// ---- DUTs/IO/Boxes/EP2008_E2806B95.TcDUT
{attribute 'GeneratedUsingTerminal: EP2008-0001-0016'}
{attribute addProperty BoxType "EP2008-0001-0016"}
{attribute addProperty Description "EP2008-0001 8 Ch. Dig. Output 24V, 0,5A, M8"}
{attribute addProperty Physics "YY"}
{attribute addProperty Id "Channel_1AT %Q*Channel_42CA91F71Channel_2AT %Q*Channel_42CA91F71Channel_3AT %Q*Channel_42CA91F71Channel_4AT %Q*Channel_42CA91F71Channel_5AT %Q*Channel_42CA91F71Channel_6AT %Q*Channel_42CA91F71Channel_7AT %Q*Channel_42CA91F71Channel_8AT %Q*Channel_42CA91F71WcStateAT %I*WcState_0B2B16F91InfoDataAT %I*InfoData_6F19DB2B2"}
{attribute addProperty CRC "3800066965"}
{attribute addProperty Size "11"}
TYPE EP2008_E2806B95 EXTENDS EtcSlaveBoxBase_77A0E4A7 :
STRUCT
	{attribute addProperty Name "Channel_1"}
	Channel_1 : Channel_42CA91F7;
	{attribute addProperty Name "Channel_2"}
	Channel_2 : Channel_42CA91F7;
	{attribute addProperty Name "Channel_3"}
	Channel_3 : Channel_42CA91F7;
	{attribute addProperty Name "Channel_4"}
	Channel_4 : Channel_42CA91F7;
	{attribute addProperty Name "Channel_5"}
	Channel_5 : Channel_42CA91F7;
	{attribute addProperty Name "Channel_6"}
	Channel_6 : Channel_42CA91F7;
	{attribute addProperty Name "Channel_7"}
	Channel_7 : Channel_42CA91F7;
	{attribute addProperty Name "Channel_8"}
	Channel_8 : Channel_42CA91F7;
	{attribute addProperty Name "WcState"}
	WcState : WcState_0B2B16F9;
	{attribute addProperty Name "InfoData"}
	InfoData : InfoData_6F19DB2B;
END_STRUCT
END_TYPE

// ---- DUTs/IO/Boxes/EP2028_E2806B95.TcDUT
{attribute 'GeneratedUsingTerminal: EP2028-0001-0016'}
{attribute addProperty BoxType "EP2028-0001-0016"}
{attribute addProperty Description "EP2028-0001 8 Ch. Dig. Output 24V, 2A, M8"}
{attribute addProperty Physics "YY"}
{attribute addProperty Id "Channel_1AT %Q*Channel_42CA91F71Channel_2AT %Q*Channel_42CA91F71Channel_3AT %Q*Channel_42CA91F71Channel_4AT %Q*Channel_42CA91F71Channel_5AT %Q*Channel_42CA91F71Channel_6AT %Q*Channel_42CA91F71Channel_7AT %Q*Channel_42CA91F71Channel_8AT %Q*Channel_42CA91F71WcStateAT %I*WcState_0B2B16F91InfoDataAT %I*InfoData_6F19DB2B2"}
{attribute addProperty CRC "3800066965"}
{attribute addProperty Size "11"}
TYPE EP2028_E2806B95 EXTENDS EtcSlaveBoxBase_77A0E4A7 :
STRUCT
	{attribute addProperty Name "Channel_1"}
	Channel_1 : Channel_42CA91F7;
	{attribute addProperty Name "Channel_2"}
	Channel_2 : Channel_42CA91F7;
	{attribute addProperty Name "Channel_3"}
	Channel_3 : Channel_42CA91F7;
	{attribute addProperty Name "Channel_4"}
	Channel_4 : Channel_42CA91F7;
	{attribute addProperty Name "Channel_5"}
	Channel_5 : Channel_42CA91F7;
	{attribute addProperty Name "Channel_6"}
	Channel_6 : Channel_42CA91F7;
	{attribute addProperty Name "Channel_7"}
	Channel_7 : Channel_42CA91F7;
	{attribute addProperty Name "Channel_8"}
	Channel_8 : Channel_42CA91F7;
	{attribute addProperty Name "WcState"}
	WcState : WcState_0B2B16F9;
	{attribute addProperty Name "InfoData"}
	InfoData : InfoData_6F19DB2B;
END_STRUCT
END_TYPE

// ---- DUTs/IO/Boxes/EP2038_3AE10DD7.TcDUT
{attribute 'GeneratedUsingTerminal: EP2038-0001-0016'}
{attribute addProperty BoxType "EP2038-0001-0016"}
{attribute addProperty Description "EP2038-0001 8 Ch. Dig. Output 24V, 2A, M8, Diagnostic"}
{attribute addProperty Physics "YY"}
{attribute addProperty Id "Diag_Channel_1AT %I*Diag_Channel_830843C11Diag_Channel_2AT %I*Diag_Channel_830843C11Diag_Channel_3AT %I*Diag_Channel_830843C11Diag_Channel_4AT %I*Diag_Channel_830843C11Diag_Channel_5AT %I*Diag_Channel_830843C11Diag_Channel_6AT %I*Diag_Channel_830843C11Diag_Channel_7AT %I*Diag_Channel_830843C11Diag_Channel_8AT %I*Diag_Channel_830843C11Channel_1AT %Q*Channel_42CA91F71Channel_2AT %Q*Channel_42CA91F71Channel_3AT %Q*Channel_42CA91F71Channel_4AT %Q*Channel_42CA91F71Channel_5AT %Q*Channel_42CA91F71Channel_6AT %Q*Channel_42CA91F71Channel_7AT %Q*Channel_42CA91F71Channel_8AT %Q*Channel_42CA91F71WcStateAT %I*WcState_9091E0EB2InfoDataAT %I*InfoData_6F19DB2B2"}
{attribute addProperty CRC "987827671"}
{attribute addProperty Size "20"}
TYPE EP2038_3AE10DD7 EXTENDS EtcSlaveBoxBase_77A0E4A7 :
STRUCT
	{attribute addProperty Name "Diag_Channel_1"}
	Diag_Channel_1 : Diag_Channel_830843C1;
	{attribute addProperty Name "Diag_Channel_2"}
	Diag_Channel_2 : Diag_Channel_830843C1;
	{attribute addProperty Name "Diag_Channel_3"}
	Diag_Channel_3 : Diag_Channel_830843C1;
	{attribute addProperty Name "Diag_Channel_4"}
	Diag_Channel_4 : Diag_Channel_830843C1;
	{attribute addProperty Name "Diag_Channel_5"}
	Diag_Channel_5 : Diag_Channel_830843C1;
	{attribute addProperty Name "Diag_Channel_6"}
	Diag_Channel_6 : Diag_Channel_830843C1;
	{attribute addProperty Name "Diag_Channel_7"}
	Diag_Channel_7 : Diag_Channel_830843C1;
	{attribute addProperty Name "Diag_Channel_8"}
	Diag_Channel_8 : Diag_Channel_830843C1;
	{attribute addProperty Name "Channel_1"}
	Channel_1 : Channel_42CA91F7;
	{attribute addProperty Name "Channel_2"}
	Channel_2 : Channel_42CA91F7;
	{attribute addProperty Name "Channel_3"}
	Channel_3 : Channel_42CA91F7;
	{attribute addProperty Name "Channel_4"}
	Channel_4 : Channel_42CA91F7;
	{attribute addProperty Name "Channel_5"}
	Channel_5 : Channel_42CA91F7;
	{attribute addProperty Name "Channel_6"}
	Channel_6 : Channel_42CA91F7;
	{attribute addProperty Name "Channel_7"}
	Channel_7 : Channel_42CA91F7;
	{attribute addProperty Name "Channel_8"}
	Channel_8 : Channel_42CA91F7;
	{attribute addProperty Name "WcState"}
	WcState : WcState_9091E0EB;
	{attribute addProperty Name "InfoData"}
	InfoData : InfoData_6F19DB2B;
END_STRUCT
END_TYPE

// ---- DUTs/IO/Boxes/EP2308_F6D9A8D1.TcDUT
{attribute 'GeneratedUsingTerminal: EP2308-0000-0016'}
{attribute addProperty BoxType "EP2308-0000-0016"}
{attribute addProperty Description "EP2308-0000 4 Ch. Dig. In, 3ms, 4 Ch. Dig. Out 24V, 0,5A, S8"}
{attribute addProperty Physics "YY"}
{attribute addProperty Id "Channel_1AT %I*Channel_830843C11Channel_2AT %I*Channel_830843C11Channel_3AT %I*Channel_830843C11Channel_4AT %I*Channel_830843C11Channel_5AT %Q*Channel_42CA91F71Channel_6AT %Q*Channel_42CA91F71Channel_7AT %Q*Channel_42CA91F71Channel_8AT %Q*Channel_42CA91F71WcStateAT %I*WcState_9091E0EB2InfoDataAT %I*InfoData_6F19DB2B2"}
{attribute addProperty CRC "4141459665"}
{attribute addProperty Size "12"}
TYPE EP2308_F6D9A8D1 EXTENDS EtcSlaveBoxBase_77A0E4A7 :
STRUCT
	{attribute addProperty Name "Channel_1"}
	Channel_1 : Channel_830843C1;
	{attribute addProperty Name "Channel_2"}
	Channel_2 : Channel_830843C1;
	{attribute addProperty Name "Channel_3"}
	Channel_3 : Channel_830843C1;
	{attribute addProperty Name "Channel_4"}
	Channel_4 : Channel_830843C1;
	{attribute addProperty Name "Channel_5"}
	Channel_5 : Channel_42CA91F7;
	{attribute addProperty Name "Channel_6"}
	Channel_6 : Channel_42CA91F7;
	{attribute addProperty Name "Channel_7"}
	Channel_7 : Channel_42CA91F7;
	{attribute addProperty Name "Channel_8"}
	Channel_8 : Channel_42CA91F7;
	{attribute addProperty Name "WcState"}
	WcState : WcState_9091E0EB;
	{attribute addProperty Name "InfoData"}
	InfoData : InfoData_6F19DB2B;
END_STRUCT
END_TYPE

// ---- DUTs/IO/Boxes/EP2316_CAC4656D.TcDUT
{attribute 'GeneratedUsingTerminal: EP2316-0003-0016'}
{attribute addProperty BoxType "EP2316-0003-0016"}
{attribute addProperty Description "EP2316-0003 8 Ch. Dig. In, 10µs, 8Ch. Dig. Out 24V, 0,5A, Diagnostic, 10-Pole Plug Connector"}
{attribute addProperty Physics "YY"}
{attribute addProperty Id "DIG_InputsAT %I*DIG_Inputs_CC4551489DIG_Diag_InputsAT %I*DIG_Diag_Inputs_584303BF8DIG_Inputs_DeviceAT %I*DIG_Inputs_Device_E94E5BF95DIG_OutputsAT %Q*DIG_Outputs_28AC1A9E8DIG_Outputs_DeviceAT %Q*DIG_Outputs_Device_36A5EF172WcStateAT %I*WcState_9091E0EB2InfoDataAT %I*InfoData_32EB74EA10"}
{attribute addProperty CRC "3401868653"}
{attribute addProperty Size "44"}
TYPE EP2316_CAC4656D EXTENDS EtcSlaveBoxBase_77A0E4A7 :
STRUCT
	{attribute addProperty Name "DIG_Inputs"}
	DIG_Inputs : DIG_Inputs_CC455148;
	{attribute addProperty Name "DIG_Diag_Inputs"}
	DIG_Diag_Inputs : DIG_Diag_Inputs_584303BF;
	{attribute addProperty Name "DIG_Inputs_Device"}
	DIG_Inputs_Device : DIG_Inputs_Device_E94E5BF9;
	{attribute addProperty Name "DIG_Outputs"}
	DIG_Outputs : DIG_Outputs_28AC1A9E;
	{attribute addProperty Name "DIG_Outputs_Device"}
	DIG_Outputs_Device : DIG_Outputs_Device_36A5EF17;
	{attribute addProperty Name "WcState"}
	WcState : WcState_9091E0EB;
	{attribute addProperty Name "InfoData"}
	InfoData : InfoData_32EB74EA;
END_STRUCT
END_TYPE

// ---- DUTs/IO/Boxes/EP2316_528F6B1F.TcDUT
{attribute 'GeneratedUsingTerminal: EP2316-0008-0016'}
{attribute addProperty BoxType "EP2316-0008-0016"}
{attribute addProperty Description "EP2316-0008 8 Ch. Dig. In, 10µs, 8Ch. Dig. Out 24V, 0,5A, Diagnostic, D-SUB25"}
{attribute addProperty Physics "YY"}
{attribute addProperty Id "DO_InputsAT %I*DO_Inputs_CC4551489DO_Diag_InputsAT %I*DO_Diag_Inputs_584303BF8DO_Inputs_DeviceAT %I*DO_Inputs_Device_AF161A9E4DO_OutputsAT %Q*DO_Outputs_28AC1A9E8DO_Outputs_DeviceAT %Q*DO_Outputs_Device_36A5EF172WcStateAT %I*WcState_9091E0EB2InfoDataAT %I*InfoData_32EB74EA10"}
{attribute addProperty CRC "1385130783"}
{attribute addProperty Size "43"}
TYPE EP2316_528F6B1F EXTENDS EtcSlaveBoxBase_77A0E4A7 :
STRUCT
	{attribute addProperty Name "DO_Inputs"}
	DO_Inputs : DO_Inputs_CC455148;
	{attribute addProperty Name "DO_Diag_Inputs"}
	DO_Diag_Inputs : DO_Diag_Inputs_584303BF;
	{attribute addProperty Name "DO_Inputs_Device"}
	DO_Inputs_Device : DO_Inputs_Device_AF161A9E;
	{attribute addProperty Name "DO_Outputs"}
	DO_Outputs : DO_Outputs_28AC1A9E;
	{attribute addProperty Name "DO_Outputs_Device"}
	DO_Outputs_Device : DO_Outputs_Device_36A5EF17;
	{attribute addProperty Name "WcState"}
	WcState : WcState_9091E0EB;
	{attribute addProperty Name "InfoData"}
	InfoData : InfoData_32EB74EA;
END_STRUCT
END_TYPE

// ---- DUTs/IO/Boxes/EP2316_3C060514.TcDUT
{attribute 'GeneratedUsingTerminal: EP2316-0008-0017'}
{attribute addProperty BoxType "EP2316-0008-0017"}
{attribute addProperty Description "EP2316-0008 8 Ch. Dig. In, 10µs, 8Ch. Dig. Out 24V, 0,5A, Diagnostic, D-SUB25"}
{attribute addProperty Physics "YY"}
{attribute addProperty Id "DO_Diag_InputsAT %I*DO_Diag_Inputs_CC4551489DO_Diag_Inputs_1AT %I*DO_Diag_Inputs_212B82C19DO_Inputs_DeviceAT %I*DO_Inputs_Device_AF161A9E4DO_OutputsAT %Q*DO_Outputs_28AC1A9E8DO_Outputs_DeviceAT %Q*DO_Outputs_Device_36A5EF172WcStateAT %I*WcState_9091E0EB2InfoDataAT %I*InfoData_32EB74EA10"}
{attribute addProperty CRC "1007027476"}
{attribute addProperty Size "44"}
TYPE EP2316_3C060514 EXTENDS EtcSlaveBoxBase_77A0E4A7 :
STRUCT
	{attribute addProperty Name "DO_Diag_Inputs"}
	DO_Diag_Inputs : DO_Diag_Inputs_CC455148;
	{attribute addProperty Name "DO_Diag_Inputs_1"}
	DO_Diag_Inputs_1 : DO_Diag_Inputs_212B82C1;
	{attribute addProperty Name "DO_Inputs_Device"}
	DO_Inputs_Device : DO_Inputs_Device_AF161A9E;
	{attribute addProperty Name "DO_Outputs"}
	DO_Outputs : DO_Outputs_28AC1A9E;
	{attribute addProperty Name "DO_Outputs_Device"}
	DO_Outputs_Device : DO_Outputs_Device_36A5EF17;
	{attribute addProperty Name "WcState"}
	WcState : WcState_9091E0EB;
	{attribute addProperty Name "InfoData"}
	InfoData : InfoData_32EB74EA;
END_STRUCT
END_TYPE

// ---- DUTs/IO/Boxes/EP2316_DCD24F8F.TcDUT
{attribute 'GeneratedUsingTerminal: EP2316-0008-0018'}
{attribute addProperty BoxType "EP2316-0008-0018"}
{attribute addProperty Description "EP2316-0008 8 Ch. Dig. In, 10µs, 8Ch. Dig. Out 24V, 0,5A, Diagnostic, D-SUB25"}
{attribute addProperty Physics "YY"}
{attribute addProperty Id "DIG_InputsAT %I*DIG_Inputs_CC4551489DIG_Diag_InputsAT %I*DIG_Diag_Inputs_584303BF8DIG_Inputs_DeviceAT %I*DIG_Inputs_Device_4E5AF17E5DIG_OutputsAT %Q*DIG_Outputs_28AC1A9E8DIG_Outputs_DeviceAT %Q*DIG_Outputs_Device_36A5EF172WcStateAT %I*WcState_9091E0EB2InfoDataAT %I*InfoData_32EB74EA10"}
{attribute addProperty CRC "3704770447"}
{attribute addProperty Size "44"}
TYPE EP2316_DCD24F8F EXTENDS EtcSlaveBoxBase_77A0E4A7 :
STRUCT
	{attribute addProperty Name "DIG_Inputs"}
	DIG_Inputs : DIG_Inputs_CC455148;
	{attribute addProperty Name "DIG_Diag_Inputs"}
	DIG_Diag_Inputs : DIG_Diag_Inputs_584303BF;
	{attribute addProperty Name "DIG_Inputs_Device"}
	DIG_Inputs_Device : DIG_Inputs_Device_4E5AF17E;
	{attribute addProperty Name "DIG_Outputs"}
	DIG_Outputs : DIG_Outputs_28AC1A9E;
	{attribute addProperty Name "DIG_Outputs_Device"}
	DIG_Outputs_Device : DIG_Outputs_Device_36A5EF17;
	{attribute addProperty Name "WcState"}
	WcState : WcState_9091E0EB;
	{attribute addProperty Name "InfoData"}
	InfoData : InfoData_32EB74EA;
END_STRUCT
END_TYPE

// ---- DUTs/IO/Boxes/EP2318_F6D9A8D1.TcDUT
{attribute 'GeneratedUsingTerminal: EP2318-0001-0016'}
{attribute addProperty BoxType "EP2318-0001-0016"}
{attribute addProperty Description "EP2318-0001 4 Ch. Dig. In, 10µs, 4 Ch. Dig. Out 24V, 0,5A, M8"}
{attribute addProperty Physics "YY"}
{attribute addProperty Id "Channel_1AT %I*Channel_830843C11Channel_2AT %I*Channel_830843C11Channel_3AT %I*Channel_830843C11Channel_4AT %I*Channel_830843C11Channel_5AT %Q*Channel_42CA91F71Channel_6AT %Q*Channel_42CA91F71Channel_7AT %Q*Channel_42CA91F71Channel_8AT %Q*Channel_42CA91F71WcStateAT %I*WcState_9091E0EB2InfoDataAT %I*InfoData_6F19DB2B2"}
{attribute addProperty CRC "4141459665"}
{attribute addProperty Size "12"}
TYPE EP2318_F6D9A8D1 EXTENDS EtcSlaveBoxBase_77A0E4A7 :
STRUCT
	{attribute addProperty Name "Channel_1"}
	Channel_1 : Channel_830843C1;
	{attribute addProperty Name "Channel_2"}
	Channel_2 : Channel_830843C1;
	{attribute addProperty Name "Channel_3"}
	Channel_3 : Channel_830843C1;
	{attribute addProperty Name "Channel_4"}
	Channel_4 : Channel_830843C1;
	{attribute addProperty Name "Channel_5"}
	Channel_5 : Channel_42CA91F7;
	{attribute addProperty Name "Channel_6"}
	Channel_6 : Channel_42CA91F7;
	{attribute addProperty Name "Channel_7"}
	Channel_7 : Channel_42CA91F7;
	{attribute addProperty Name "Channel_8"}
	Channel_8 : Channel_42CA91F7;
	{attribute addProperty Name "WcState"}
	WcState : WcState_9091E0EB;
	{attribute addProperty Name "InfoData"}
	InfoData : InfoData_6F19DB2B;
END_STRUCT
END_TYPE

// ---- DUTs/IO/Boxes/EP2328_F6D9A8D1.TcDUT
{attribute 'GeneratedUsingTerminal: EP2328-0001-0016'}
{attribute addProperty BoxType "EP2328-0001-0016"}
{attribute addProperty Description "EP2328-0001 4 CH. Dig. In, 3ms, 4 Ch. Dig. Out 24V, 2A, M8"}
{attribute addProperty Physics "YY"}
{attribute addProperty Id "Channel_1AT %I*Channel_830843C11Channel_2AT %I*Channel_830843C11Channel_3AT %I*Channel_830843C11Channel_4AT %I*Channel_830843C11Channel_5AT %Q*Channel_42CA91F71Channel_6AT %Q*Channel_42CA91F71Channel_7AT %Q*Channel_42CA91F71Channel_8AT %Q*Channel_42CA91F71WcStateAT %I*WcState_9091E0EB2InfoDataAT %I*InfoData_6F19DB2B2"}
{attribute addProperty CRC "4141459665"}
{attribute addProperty Size "12"}
TYPE EP2328_F6D9A8D1 EXTENDS EtcSlaveBoxBase_77A0E4A7 :
STRUCT
	{attribute addProperty Name "Channel_1"}
	Channel_1 : Channel_830843C1;
	{attribute addProperty Name "Channel_2"}
	Channel_2 : Channel_830843C1;
	{attribute addProperty Name "Channel_3"}
	Channel_3 : Channel_830843C1;
	{attribute addProperty Name "Channel_4"}
	Channel_4 : Channel_830843C1;
	{attribute addProperty Name "Channel_5"}
	Channel_5 : Channel_42CA91F7;
	{attribute addProperty Name "Channel_6"}
	Channel_6 : Channel_42CA91F7;
	{attribute addProperty Name "Channel_7"}
	Channel_7 : Channel_42CA91F7;
	{attribute addProperty Name "Channel_8"}
	Channel_8 : Channel_42CA91F7;
	{attribute addProperty Name "WcState"}
	WcState : WcState_9091E0EB;
	{attribute addProperty Name "InfoData"}
	InfoData : InfoData_6F19DB2B;
END_STRUCT
END_TYPE

// ---- DUTs/IO/Boxes/EP2328_F66CDDB7.TcDUT
{attribute 'GeneratedUsingTerminal: EP2328-1061-0016'}
{attribute addProperty BoxType "EP2328-1061-0016"}
{attribute addProperty Description "EP2328-1061 4 Ch. Dig. In, 10µs, 4 Ch. Dig. Out 24V, 2A, M8 cable"}
{attribute addProperty Physics "YY"}
{attribute addProperty Id "DI_X01_Pin4_InputAT %I*DI_X01_Pin4_Input_830843C11DI_X01_Pin2_InputAT %I*DI_X01_Pin2_Input_830843C11DI_X02_Pin4_InputAT %I*DI_X02_Pin4_Input_830843C11DI_X02_Pin2_InputAT %I*DI_X02_Pin2_Input_830843C11DO_X03_Pin4_OutputAT %Q*DO_X03_Pin4_Output_42CA91F71DO_X03_Pin2_OutputAT %Q*DO_X03_Pin2_Output_42CA91F71DO_X04_Pin4_OutputAT %Q*DO_X04_Pin4_Output_42CA91F71DO_X04_Pin2_OutputAT %Q*DO_X04_Pin2_Output_42CA91F71WcStateAT %I*WcState_9091E0EB2InfoDataAT %I*InfoData_6F19DB2B2"}
{attribute addProperty CRC "4134329783"}
{attribute addProperty Size "12"}
TYPE EP2328_F66CDDB7 EXTENDS EtcSlaveBoxBase_77A0E4A7 :
STRUCT
	{attribute addProperty Name "DI_X01_Pin4_Input"}
	DI_X01_Pin4_Input : DI_X01_Pin4_Input_830843C1;
	{attribute addProperty Name "DI_X01_Pin2_Input"}
	DI_X01_Pin2_Input : DI_X01_Pin2_Input_830843C1;
	{attribute addProperty Name "DI_X02_Pin4_Input"}
	DI_X02_Pin4_Input : DI_X02_Pin4_Input_830843C1;
	{attribute addProperty Name "DI_X02_Pin2_Input"}
	DI_X02_Pin2_Input : DI_X02_Pin2_Input_830843C1;
	{attribute addProperty Name "DO_X03_Pin4_Output"}
	DO_X03_Pin4_Output : DO_X03_Pin4_Output_42CA91F7;
	{attribute addProperty Name "DO_X03_Pin2_Output"}
	DO_X03_Pin2_Output : DO_X03_Pin2_Output_42CA91F7;
	{attribute addProperty Name "DO_X04_Pin4_Output"}
	DO_X04_Pin4_Output : DO_X04_Pin4_Output_42CA91F7;
	{attribute addProperty Name "DO_X04_Pin2_Output"}
	DO_X04_Pin2_Output : DO_X04_Pin2_Output_42CA91F7;
	{attribute addProperty Name "WcState"}
	WcState : WcState_9091E0EB;
	{attribute addProperty Name "InfoData"}
	InfoData : InfoData_6F19DB2B;
END_STRUCT
END_TYPE

// ---- DUTs/IO/Boxes/EP2338_39FFBC52.TcDUT
{attribute 'GeneratedUsingTerminal: EP2338-0001-0016'}
{attribute addProperty BoxType "EP2338-0001-0016"}
{attribute addProperty Description "EP2338-0001 8 Ch. Dig. Input/Output 24V, 0,5A, M8"}
{attribute addProperty Physics "YY"}
{attribute addProperty Id "Channel_1AT %I*Channel_830843C11Channel_2AT %I*Channel_830843C11Channel_3AT %I*Channel_830843C11Channel_4AT %I*Channel_830843C11Channel_5AT %I*Channel_830843C11Channel_6AT %I*Channel_830843C11Channel_7AT %I*Channel_830843C11Channel_8AT %I*Channel_830843C11Channel_1_1AT %Q*Channel_42CA91F71Channel_2_1AT %Q*Channel_42CA91F71Channel_3_1AT %Q*Channel_42CA91F71Channel_4_1AT %Q*Channel_42CA91F71Channel_5_1AT %Q*Channel_42CA91F71Channel_6_1AT %Q*Channel_42CA91F71Channel_7_1AT %Q*Channel_42CA91F71Channel_8_1AT %Q*Channel_42CA91F71WcStateAT %I*WcState_9091E0EB2InfoDataAT %I*InfoData_6F19DB2B2"}
{attribute addProperty CRC "973061202"}
{attribute addProperty Size "20"}
TYPE EP2338_39FFBC52 EXTENDS EtcSlaveBoxBase_77A0E4A7 :
STRUCT
	{attribute addProperty Name "Channel_1"}
	Channel_1 : Channel_830843C1;
	{attribute addProperty Name "Channel_2"}
	Channel_2 : Channel_830843C1;
	{attribute addProperty Name "Channel_3"}
	Channel_3 : Channel_830843C1;
	{attribute addProperty Name "Channel_4"}
	Channel_4 : Channel_830843C1;
	{attribute addProperty Name "Channel_5"}
	Channel_5 : Channel_830843C1;
	{attribute addProperty Name "Channel_6"}
	Channel_6 : Channel_830843C1;
	{attribute addProperty Name "Channel_7"}
	Channel_7 : Channel_830843C1;
	{attribute addProperty Name "Channel_8"}
	Channel_8 : Channel_830843C1;
	{attribute addProperty Name "Channel_1_1"}
	Channel_1_1 : Channel_42CA91F7;
	{attribute addProperty Name "Channel_2_1"}
	Channel_2_1 : Channel_42CA91F7;
	{attribute addProperty Name "Channel_3_1"}
	Channel_3_1 : Channel_42CA91F7;
	{attribute addProperty Name "Channel_4_1"}
	Channel_4_1 : Channel_42CA91F7;
	{attribute addProperty Name "Channel_5_1"}
	Channel_5_1 : Channel_42CA91F7;
	{attribute addProperty Name "Channel_6_1"}
	Channel_6_1 : Channel_42CA91F7;
	{attribute addProperty Name "Channel_7_1"}
	Channel_7_1 : Channel_42CA91F7;
	{attribute addProperty Name "Channel_8_1"}
	Channel_8_1 : Channel_42CA91F7;
	{attribute addProperty Name "WcState"}
	WcState : WcState_9091E0EB;
	{attribute addProperty Name "InfoData"}
	InfoData : InfoData_6F19DB2B;
END_STRUCT
END_TYPE

// ---- DUTs/IO/Boxes/EP2338_7699BCF6.TcDUT
{attribute 'GeneratedUsingTerminal: EP2338-0001-0018'}
{attribute addProperty BoxType "EP2338-0001-0018"}
{attribute addProperty Description "EP2338-0001 8 Ch. Dig. Input/Output 24V, 0,5A, M8"}
{attribute addProperty Physics "YY"}
{attribute addProperty Id "Channel_1AT %I*Channel_830843C11Channel_2AT %I*Channel_830843C11Channel_3AT %I*Channel_830843C11Channel_4AT %I*Channel_830843C11Channel_5AT %I*Channel_830843C11Channel_6AT %I*Channel_830843C11Channel_7AT %I*Channel_830843C11Channel_8AT %I*Channel_830843C11Channel_9AT %Q*Channel_42CA91F71Channel_10AT %Q*Channel_42CA91F71Channel_11AT %Q*Channel_42CA91F71Channel_12AT %Q*Channel_42CA91F71Channel_13AT %Q*Channel_42CA91F71Channel_14AT %Q*Channel_42CA91F71Channel_15AT %Q*Channel_42CA91F71Channel_16AT %Q*Channel_42CA91F71WcStateAT %I*WcState_9091E0EB2InfoDataAT %I*InfoData_6F19DB2B2"}
{attribute addProperty CRC "1989786870"}
{attribute addProperty Size "20"}
TYPE EP2338_7699BCF6 EXTENDS EtcSlaveBoxBase_77A0E4A7 :
STRUCT
	{attribute addProperty Name "Channel_1"}
	Channel_1 : Channel_830843C1;
	{attribute addProperty Name "Channel_2"}
	Channel_2 : Channel_830843C1;
	{attribute addProperty Name "Channel_3"}
	Channel_3 : Channel_830843C1;
	{attribute addProperty Name "Channel_4"}
	Channel_4 : Channel_830843C1;
	{attribute addProperty Name "Channel_5"}
	Channel_5 : Channel_830843C1;
	{attribute addProperty Name "Channel_6"}
	Channel_6 : Channel_830843C1;
	{attribute addProperty Name "Channel_7"}
	Channel_7 : Channel_830843C1;
	{attribute addProperty Name "Channel_8"}
	Channel_8 : Channel_830843C1;
	{attribute addProperty Name "Channel_9"}
	Channel_9 : Channel_42CA91F7;
	{attribute addProperty Name "Channel_10"}
	Channel_10 : Channel_42CA91F7;
	{attribute addProperty Name "Channel_11"}
	Channel_11 : Channel_42CA91F7;
	{attribute addProperty Name "Channel_12"}
	Channel_12 : Channel_42CA91F7;
	{attribute addProperty Name "Channel_13"}
	Channel_13 : Channel_42CA91F7;
	{attribute addProperty Name "Channel_14"}
	Channel_14 : Channel_42CA91F7;
	{attribute addProperty Name "Channel_15"}
	Channel_15 : Channel_42CA91F7;
	{attribute addProperty Name "Channel_16"}
	Channel_16 : Channel_42CA91F7;
	{attribute addProperty Name "WcState"}
	WcState : WcState_9091E0EB;
	{attribute addProperty Name "InfoData"}
	InfoData : InfoData_6F19DB2B;
END_STRUCT
END_TYPE

// ---- DUTs/IO/Boxes/EP2339_B2B612E8.TcDUT
{attribute 'GeneratedUsingTerminal: EP2339-0003-0016'}
{attribute addProperty BoxType "EP2339-0003-0016"}
{attribute addProperty Description "EP2339-0003 16 Ch. Dig. Input/Output 24V, 0,5A, 10-Pole Plug Connector"}
{attribute addProperty Physics "YY"}
{attribute addProperty Id "DI_Inputs_Channel_1AT %I*DI_Inputs_Channel_91AC31B711DI_Inputs_Channel_2AT %I*DI_Inputs_Channel_91AC31B711DO_Outputs_Channel_1AT %Q*DO_Outputs_Channel_28AC1A9E8DO_Outputs_Channel_2AT %Q*DO_Outputs_Channel_28AC1A9E8WcStateAT %I*WcState_9091E0EB2InfoDataAT %I*InfoData_32EB74EA10"}
{attribute addProperty CRC "2998276840"}
{attribute addProperty Size "50"}
TYPE EP2339_B2B612E8 EXTENDS EtcSlaveBoxBase_77A0E4A7 :
STRUCT
	{attribute addProperty Name "DI_Inputs_Channel_1"}
	DI_Inputs_Channel_1 : DI_Inputs_Channel_91AC31B7;
	{attribute addProperty Name "DI_Inputs_Channel_2"}
	DI_Inputs_Channel_2 : DI_Inputs_Channel_91AC31B7;
	{attribute addProperty Name "DO_Outputs_Channel_1"}
	DO_Outputs_Channel_1 : DO_Outputs_Channel_28AC1A9E;
	{attribute addProperty Name "DO_Outputs_Channel_2"}
	DO_Outputs_Channel_2 : DO_Outputs_Channel_28AC1A9E;
	{attribute addProperty Name "WcState"}
	WcState : WcState_9091E0EB;
	{attribute addProperty Name "InfoData"}
	InfoData : InfoData_32EB74EA;
END_STRUCT
END_TYPE

// ---- DUTs/IO/Boxes/EP2339_C2A6198C.TcDUT
{attribute 'GeneratedUsingTerminal: EP2339-0021-0016'}
{attribute addProperty BoxType "EP2339-0021-0016"}
{attribute addProperty Description "EP2339-0021 16 Ch. Dig. Input/Output 24V, 0,5A, M8"}
{attribute addProperty Physics "YY"}
{attribute addProperty Id "Channel_1AT %I*Channel_830843C11Channel_2AT %I*Channel_830843C11Channel_3AT %I*Channel_830843C11Channel_4AT %I*Channel_830843C11Channel_5AT %I*Channel_830843C11Channel_6AT %I*Channel_830843C11Channel_7AT %I*Channel_830843C11Channel_8AT %I*Channel_830843C11Channel_9AT %I*Channel_830843C11Channel_10AT %I*Channel_830843C11Channel_11AT %I*Channel_830843C11Channel_12AT %I*Channel_830843C11Channel_13AT %I*Channel_830843C11Channel_14AT %I*Channel_830843C11Channel_15AT %I*Channel_830843C11Channel_16AT %I*Channel_830843C11Channel_1_1AT %Q*Channel_42CA91F71Channel_2_1AT %Q*Channel_42CA91F71Channel_3_1AT %Q*Channel_42CA91F71Channel_4_1AT %Q*Channel_42CA91F71Channel_5_1AT %Q*Channel_42CA91F71Channel_6_1AT %Q*Channel_42CA91F71Channel_7_1AT %Q*Channel_42CA91F71Channel_8_1AT %Q*Channel_42CA91F71Channel_9_1AT %Q*Channel_42CA91F71Channel_10_1AT %Q*Channel_42CA91F71Channel_11_1AT %Q*Channel_42CA91F71Channel_12_1AT %Q*Channel_42CA91F71Channel_13_1AT %Q*Channel_42CA91F71Channel_14_1AT %Q*Channel_42CA91F71Channel_15_1AT %Q*Channel_42CA91F71Channel_16_1AT %Q*Channel_42CA91F71WcStateAT %I*WcState_9091E0EB2InfoDataAT %I*InfoData_0A66F0098"}
{attribute addProperty CRC "3265665420"}
{attribute addProperty Size "42"}
TYPE EP2339_C2A6198C EXTENDS EtcSlaveBoxBase_77A0E4A7 :
STRUCT
	{attribute addProperty Name "Channel_1"}
	Channel_1 : Channel_830843C1;
	{attribute addProperty Name "Channel_2"}
	Channel_2 : Channel_830843C1;
	{attribute addProperty Name "Channel_3"}
	Channel_3 : Channel_830843C1;
	{attribute addProperty Name "Channel_4"}
	Channel_4 : Channel_830843C1;
	{attribute addProperty Name "Channel_5"}
	Channel_5 : Channel_830843C1;
	{attribute addProperty Name "Channel_6"}
	Channel_6 : Channel_830843C1;
	{attribute addProperty Name "Channel_7"}
	Channel_7 : Channel_830843C1;
	{attribute addProperty Name "Channel_8"}
	Channel_8 : Channel_830843C1;
	{attribute addProperty Name "Channel_9"}
	Channel_9 : Channel_830843C1;
	{attribute addProperty Name "Channel_10"}
	Channel_10 : Channel_830843C1;
	{attribute addProperty Name "Channel_11"}
	Channel_11 : Channel_830843C1;
	{attribute addProperty Name "Channel_12"}
	Channel_12 : Channel_830843C1;
	{attribute addProperty Name "Channel_13"}
	Channel_13 : Channel_830843C1;
	{attribute addProperty Name "Channel_14"}
	Channel_14 : Channel_830843C1;
	{attribute addProperty Name "Channel_15"}
	Channel_15 : Channel_830843C1;
	{attribute addProperty Name "Channel_16"}
	Channel_16 : Channel_830843C1;
	{attribute addProperty Name "Channel_1_1"}
	Channel_1_1 : Channel_42CA91F7;
	{attribute addProperty Name "Channel_2_1"}
	Channel_2_1 : Channel_42CA91F7;
	{attribute addProperty Name "Channel_3_1"}
	Channel_3_1 : Channel_42CA91F7;
	{attribute addProperty Name "Channel_4_1"}
	Channel_4_1 : Channel_42CA91F7;
	{attribute addProperty Name "Channel_5_1"}
	Channel_5_1 : Channel_42CA91F7;
	{attribute addProperty Name "Channel_6_1"}
	Channel_6_1 : Channel_42CA91F7;
	{attribute addProperty Name "Channel_7_1"}
	Channel_7_1 : Channel_42CA91F7;
	{attribute addProperty Name "Channel_8_1"}
	Channel_8_1 : Channel_42CA91F7;
	{attribute addProperty Name "Channel_9_1"}
	Channel_9_1 : Channel_42CA91F7;
	{attribute addProperty Name "Channel_10_1"}
	Channel_10_1 : Channel_42CA91F7;
	{attribute addProperty Name "Channel_11_1"}
	Channel_11_1 : Channel_42CA91F7;
	{attribute addProperty Name "Channel_12_1"}
	Channel_12_1 : Channel_42CA91F7;
	{attribute addProperty Name "Channel_13_1"}
	Channel_13_1 : Channel_42CA91F7;
	{attribute addProperty Name "Channel_14_1"}
	Channel_14_1 : Channel_42CA91F7;
	{attribute addProperty Name "Channel_15_1"}
	Channel_15_1 : Channel_42CA91F7;
	{attribute addProperty Name "Channel_16_1"}
	Channel_16_1 : Channel_42CA91F7;
	{attribute addProperty Name "WcState"}
	WcState : WcState_9091E0EB;
	{attribute addProperty Name "InfoData"}
	InfoData : InfoData_0A66F009;
END_STRUCT
END_TYPE

// ---- DUTs/IO/Boxes/EP2339_D8E9F29A.TcDUT
{attribute 'GeneratedUsingTerminal: EP2339-0021-0017'}
{attribute addProperty BoxType "EP2339-0021-0017"}
{attribute addProperty Description "EP2339-0021 16 Ch. Dig. Input/Output 24V, 0,5A, M8"}
{attribute addProperty Physics "YY"}
{attribute addProperty Id "Channel_1AT %I*Channel_830843C11Channel_2AT %I*Channel_830843C11Channel_3AT %I*Channel_830843C11Channel_4AT %I*Channel_830843C11Channel_5AT %I*Channel_830843C11Channel_6AT %I*Channel_830843C11Channel_7AT %I*Channel_830843C11Channel_8AT %I*Channel_830843C11Channel_9AT %I*Channel_830843C11Channel_10AT %I*Channel_830843C11Channel_11AT %I*Channel_830843C11Channel_12AT %I*Channel_830843C11Channel_13AT %I*Channel_830843C11Channel_14AT %I*Channel_830843C11Channel_15AT %I*Channel_830843C11Channel_16AT %I*Channel_830843C11Channel_17AT %Q*Channel_42CA91F71Channel_18AT %Q*Channel_42CA91F71Channel_19AT %Q*Channel_42CA91F71Channel_20AT %Q*Channel_42CA91F71Channel_21AT %Q*Channel_42CA91F71Channel_22AT %Q*Channel_42CA91F71Channel_23AT %Q*Channel_42CA91F71Channel_24AT %Q*Channel_42CA91F71Channel_25AT %Q*Channel_42CA91F71Channel_26AT %Q*Channel_42CA91F71Channel_27AT %Q*Channel_42CA91F71Channel_28AT %Q*Channel_42CA91F71Channel_29AT %Q*Channel_42CA91F71Channel_30AT %Q*Channel_42CA91F71Channel_31AT %Q*Channel_42CA91F71Channel_32AT %Q*Channel_42CA91F71WcStateAT %I*WcState_9091E0EB2InfoDataAT %I*InfoData_0A66F0098"}
{attribute addProperty CRC "3639210650"}
{attribute addProperty Size "42"}
TYPE EP2339_D8E9F29A EXTENDS EtcSlaveBoxBase_77A0E4A7 :
STRUCT
	{attribute addProperty Name "Channel_1"}
	Channel_1 : Channel_830843C1;
	{attribute addProperty Name "Channel_2"}
	Channel_2 : Channel_830843C1;
	{attribute addProperty Name "Channel_3"}
	Channel_3 : Channel_830843C1;
	{attribute addProperty Name "Channel_4"}
	Channel_4 : Channel_830843C1;
	{attribute addProperty Name "Channel_5"}
	Channel_5 : Channel_830843C1;
	{attribute addProperty Name "Channel_6"}
	Channel_6 : Channel_830843C1;
	{attribute addProperty Name "Channel_7"}
	Channel_7 : Channel_830843C1;
	{attribute addProperty Name "Channel_8"}
	Channel_8 : Channel_830843C1;
	{attribute addProperty Name "Channel_9"}
	Channel_9 : Channel_830843C1;
	{attribute addProperty Name "Channel_10"}
	Channel_10 : Channel_830843C1;
	{attribute addProperty Name "Channel_11"}
	Channel_11 : Channel_830843C1;
	{attribute addProperty Name "Channel_12"}
	Channel_12 : Channel_830843C1;
	{attribute addProperty Name "Channel_13"}
	Channel_13 : Channel_830843C1;
	{attribute addProperty Name "Channel_14"}
	Channel_14 : Channel_830843C1;
	{attribute addProperty Name "Channel_15"}
	Channel_15 : Channel_830843C1;
	{attribute addProperty Name "Channel_16"}
	Channel_16 : Channel_830843C1;
	{attribute addProperty Name "Channel_17"}
	Channel_17 : Channel_42CA91F7;
	{attribute addProperty Name "Channel_18"}
	Channel_18 : Channel_42CA91F7;
	{attribute addProperty Name "Channel_19"}
	Channel_19 : Channel_42CA91F7;
	{attribute addProperty Name "Channel_20"}
	Channel_20 : Channel_42CA91F7;
	{attribute addProperty Name "Channel_21"}
	Channel_21 : Channel_42CA91F7;
	{attribute addProperty Name "Channel_22"}
	Channel_22 : Channel_42CA91F7;
	{attribute addProperty Name "Channel_23"}
	Channel_23 : Channel_42CA91F7;
	{attribute addProperty Name "Channel_24"}
	Channel_24 : Channel_42CA91F7;
	{attribute addProperty Name "Channel_25"}
	Channel_25 : Channel_42CA91F7;
	{attribute addProperty Name "Channel_26"}
	Channel_26 : Channel_42CA91F7;
	{attribute addProperty Name "Channel_27"}
	Channel_27 : Channel_42CA91F7;
	{attribute addProperty Name "Channel_28"}
	Channel_28 : Channel_42CA91F7;
	{attribute addProperty Name "Channel_29"}
	Channel_29 : Channel_42CA91F7;
	{attribute addProperty Name "Channel_30"}
	Channel_30 : Channel_42CA91F7;
	{attribute addProperty Name "Channel_31"}
	Channel_31 : Channel_42CA91F7;
	{attribute addProperty Name "Channel_32"}
	Channel_32 : Channel_42CA91F7;
	{attribute addProperty Name "WcState"}
	WcState : WcState_9091E0EB;
	{attribute addProperty Name "InfoData"}
	InfoData : InfoData_0A66F009;
END_STRUCT
END_TYPE

// ---- DUTs/IO/Boxes/EP2339_4CF33DED.TcDUT
{attribute 'GeneratedUsingTerminal: EP2339-0021-0019'}
{attribute addProperty BoxType "EP2339-0021-0019"}
{attribute addProperty Description "EP2339-0021 16 Ch. Dig. Input/Output 24V, 0,5A, M8"}
{attribute addProperty Physics "YY"}
{attribute addProperty Id "Channel_1AT %I*Channel_830843C11Channel_2AT %I*Channel_830843C11Channel_3AT %I*Channel_830843C11Channel_4AT %I*Channel_830843C11Channel_5AT %I*Channel_830843C11Channel_6AT %I*Channel_830843C11Channel_7AT %I*Channel_830843C11Channel_8AT %I*Channel_830843C11Channel_9AT %I*Channel_830843C11Channel_10AT %I*Channel_830843C11Channel_11AT %I*Channel_830843C11Channel_12AT %I*Channel_830843C11Channel_13AT %I*Channel_830843C11Channel_14AT %I*Channel_830843C11Channel_15AT %I*Channel_830843C11Channel_16AT %I*Channel_830843C11Channel_17AT %Q*Channel_42CA91F71Channel_18AT %Q*Channel_42CA91F71Channel_19AT %Q*Channel_42CA91F71Channel_20AT %Q*Channel_42CA91F71Channel_21AT %Q*Channel_42CA91F71Channel_22AT %Q*Channel_42CA91F71Channel_23AT %Q*Channel_42CA91F71Channel_24AT %Q*Channel_42CA91F71Channel_25AT %Q*Channel_42CA91F71Channel_26AT %Q*Channel_42CA91F71Channel_27AT %Q*Channel_42CA91F71Channel_28AT %Q*Channel_42CA91F71Channel_29AT %Q*Channel_42CA91F71Channel_30AT %Q*Channel_42CA91F71Channel_31AT %Q*Channel_42CA91F71Channel_32AT %Q*Channel_42CA91F71WcStateAT %I*WcState_9091E0EB2InfoDataAT %I*InfoData_6F19DB2B2"}
{attribute addProperty CRC "1291009517"}
{attribute addProperty Size "36"}
TYPE EP2339_4CF33DED EXTENDS EtcSlaveBoxBase_77A0E4A7 :
STRUCT
	{attribute addProperty Name "Channel_1"}
	Channel_1 : Channel_830843C1;
	{attribute addProperty Name "Channel_2"}
	Channel_2 : Channel_830843C1;
	{attribute addProperty Name "Channel_3"}
	Channel_3 : Channel_830843C1;
	{attribute addProperty Name "Channel_4"}
	Channel_4 : Channel_830843C1;
	{attribute addProperty Name "Channel_5"}
	Channel_5 : Channel_830843C1;
	{attribute addProperty Name "Channel_6"}
	Channel_6 : Channel_830843C1;
	{attribute addProperty Name "Channel_7"}
	Channel_7 : Channel_830843C1;
	{attribute addProperty Name "Channel_8"}
	Channel_8 : Channel_830843C1;
	{attribute addProperty Name "Channel_9"}
	Channel_9 : Channel_830843C1;
	{attribute addProperty Name "Channel_10"}
	Channel_10 : Channel_830843C1;
	{attribute addProperty Name "Channel_11"}
	Channel_11 : Channel_830843C1;
	{attribute addProperty Name "Channel_12"}
	Channel_12 : Channel_830843C1;
	{attribute addProperty Name "Channel_13"}
	Channel_13 : Channel_830843C1;
	{attribute addProperty Name "Channel_14"}
	Channel_14 : Channel_830843C1;
	{attribute addProperty Name "Channel_15"}
	Channel_15 : Channel_830843C1;
	{attribute addProperty Name "Channel_16"}
	Channel_16 : Channel_830843C1;
	{attribute addProperty Name "Channel_17"}
	Channel_17 : Channel_42CA91F7;
	{attribute addProperty Name "Channel_18"}
	Channel_18 : Channel_42CA91F7;
	{attribute addProperty Name "Channel_19"}
	Channel_19 : Channel_42CA91F7;
	{attribute addProperty Name "Channel_20"}
	Channel_20 : Channel_42CA91F7;
	{attribute addProperty Name "Channel_21"}
	Channel_21 : Channel_42CA91F7;
	{attribute addProperty Name "Channel_22"}
	Channel_22 : Channel_42CA91F7;
	{attribute addProperty Name "Channel_23"}
	Channel_23 : Channel_42CA91F7;
	{attribute addProperty Name "Channel_24"}
	Channel_24 : Channel_42CA91F7;
	{attribute addProperty Name "Channel_25"}
	Channel_25 : Channel_42CA91F7;
	{attribute addProperty Name "Channel_26"}
	Channel_26 : Channel_42CA91F7;
	{attribute addProperty Name "Channel_27"}
	Channel_27 : Channel_42CA91F7;
	{attribute addProperty Name "Channel_28"}
	Channel_28 : Channel_42CA91F7;
	{attribute addProperty Name "Channel_29"}
	Channel_29 : Channel_42CA91F7;
	{attribute addProperty Name "Channel_30"}
	Channel_30 : Channel_42CA91F7;
	{attribute addProperty Name "Channel_31"}
	Channel_31 : Channel_42CA91F7;
	{attribute addProperty Name "Channel_32"}
	Channel_32 : Channel_42CA91F7;
	{attribute addProperty Name "WcState"}
	WcState : WcState_9091E0EB;
	{attribute addProperty Name "InfoData"}
	InfoData : InfoData_6F19DB2B;
END_STRUCT
END_TYPE

// ---- DUTs/IO/Boxes/EP2339_56BCD6FB.TcDUT
{attribute 'GeneratedUsingTerminal: EP2339-0022-0016'}
{attribute addProperty BoxType "EP2339-0022-0016"}
{attribute addProperty Description "EP2339-0022 16 Ch. Dig. Input/Output 24V, 0,5A, M12"}
{attribute addProperty Physics "YY"}
{attribute addProperty Id "Channel_1AT %I*Channel_830843C11Channel_2AT %I*Channel_830843C11Channel_3AT %I*Channel_830843C11Channel_4AT %I*Channel_830843C11Channel_5AT %I*Channel_830843C11Channel_6AT %I*Channel_830843C11Channel_7AT %I*Channel_830843C11Channel_8AT %I*Channel_830843C11Channel_9AT %I*Channel_830843C11Channel_10AT %I*Channel_830843C11Channel_11AT %I*Channel_830843C11Channel_12AT %I*Channel_830843C11Channel_13AT %I*Channel_830843C11Channel_14AT %I*Channel_830843C11Channel_15AT %I*Channel_830843C11Channel_16AT %I*Channel_830843C11Channel_1_1AT %Q*Channel_42CA91F71Channel_2_1AT %Q*Channel_42CA91F71Channel_3_1AT %Q*Channel_42CA91F71Channel_4_1AT %Q*Channel_42CA91F71Channel_5_1AT %Q*Channel_42CA91F71Channel_6_1AT %Q*Channel_42CA91F71Channel_7_1AT %Q*Channel_42CA91F71Channel_8_1AT %Q*Channel_42CA91F71Channel_9_1AT %Q*Channel_42CA91F71Channel_10_1AT %Q*Channel_42CA91F71Channel_11_1AT %Q*Channel_42CA91F71Channel_12_1AT %Q*Channel_42CA91F71Channel_13_1AT %Q*Channel_42CA91F71Channel_14_1AT %Q*Channel_42CA91F71Channel_15_1AT %Q*Channel_42CA91F71Channel_16_1AT %Q*Channel_42CA91F71WcStateAT %I*WcState_9091E0EB2InfoDataAT %I*InfoData_6F19DB2B2"}
{attribute addProperty CRC "1455216379"}
{attribute addProperty Size "36"}
TYPE EP2339_56BCD6FB EXTENDS EtcSlaveBoxBase_77A0E4A7 :
STRUCT
	{attribute addProperty Name "Channel_1"}
	Channel_1 : Channel_830843C1;
	{attribute addProperty Name "Channel_2"}
	Channel_2 : Channel_830843C1;
	{attribute addProperty Name "Channel_3"}
	Channel_3 : Channel_830843C1;
	{attribute addProperty Name "Channel_4"}
	Channel_4 : Channel_830843C1;
	{attribute addProperty Name "Channel_5"}
	Channel_5 : Channel_830843C1;
	{attribute addProperty Name "Channel_6"}
	Channel_6 : Channel_830843C1;
	{attribute addProperty Name "Channel_7"}
	Channel_7 : Channel_830843C1;
	{attribute addProperty Name "Channel_8"}
	Channel_8 : Channel_830843C1;
	{attribute addProperty Name "Channel_9"}
	Channel_9 : Channel_830843C1;
	{attribute addProperty Name "Channel_10"}
	Channel_10 : Channel_830843C1;
	{attribute addProperty Name "Channel_11"}
	Channel_11 : Channel_830843C1;
	{attribute addProperty Name "Channel_12"}
	Channel_12 : Channel_830843C1;
	{attribute addProperty Name "Channel_13"}
	Channel_13 : Channel_830843C1;
	{attribute addProperty Name "Channel_14"}
	Channel_14 : Channel_830843C1;
	{attribute addProperty Name "Channel_15"}
	Channel_15 : Channel_830843C1;
	{attribute addProperty Name "Channel_16"}
	Channel_16 : Channel_830843C1;
	{attribute addProperty Name "Channel_1_1"}
	Channel_1_1 : Channel_42CA91F7;
	{attribute addProperty Name "Channel_2_1"}
	Channel_2_1 : Channel_42CA91F7;
	{attribute addProperty Name "Channel_3_1"}
	Channel_3_1 : Channel_42CA91F7;
	{attribute addProperty Name "Channel_4_1"}
	Channel_4_1 : Channel_42CA91F7;
	{attribute addProperty Name "Channel_5_1"}
	Channel_5_1 : Channel_42CA91F7;
	{attribute addProperty Name "Channel_6_1"}
	Channel_6_1 : Channel_42CA91F7;
	{attribute addProperty Name "Channel_7_1"}
	Channel_7_1 : Channel_42CA91F7;
	{attribute addProperty Name "Channel_8_1"}
	Channel_8_1 : Channel_42CA91F7;
	{attribute addProperty Name "Channel_9_1"}
	Channel_9_1 : Channel_42CA91F7;
	{attribute addProperty Name "Channel_10_1"}
	Channel_10_1 : Channel_42CA91F7;
	{attribute addProperty Name "Channel_11_1"}
	Channel_11_1 : Channel_42CA91F7;
	{attribute addProperty Name "Channel_12_1"}
	Channel_12_1 : Channel_42CA91F7;
	{attribute addProperty Name "Channel_13_1"}
	Channel_13_1 : Channel_42CA91F7;
	{attribute addProperty Name "Channel_14_1"}
	Channel_14_1 : Channel_42CA91F7;
	{attribute addProperty Name "Channel_15_1"}
	Channel_15_1 : Channel_42CA91F7;
	{attribute addProperty Name "Channel_16_1"}
	Channel_16_1 : Channel_42CA91F7;
	{attribute addProperty Name "WcState"}
	WcState : WcState_9091E0EB;
	{attribute addProperty Name "InfoData"}
	InfoData : InfoData_6F19DB2B;
END_STRUCT
END_TYPE

// ---- DUTs/IO/Boxes/EP2339_49541507.TcDUT
{attribute 'GeneratedUsingTerminal: EP2339-0042-0017'}
{attribute addProperty BoxType "EP2339-0042-0017"}
{attribute addProperty Description "EP2339-0042 16 Ch. Dig. Input/Output 24V, 0.5A, M12 "}
{attribute addProperty Physics "YY"}
{attribute addProperty Id "DI_X01_Pin4AT %I*DI_X01_Pin_830843C11DI_X01_Pin2AT %I*DI_X01_Pin_830843C11DI_X02_Pin4AT %I*DI_X02_Pin_830843C11DI_X02_Pin2AT %I*DI_X02_Pin_830843C11DI_X03_Pin4AT %I*DI_X03_Pin_830843C11DI_X03_Pin2AT %I*DI_X03_Pin_830843C11DI_X04_Pin4AT %I*DI_X04_Pin_830843C11DI_X04_Pin2AT %I*DI_X04_Pin_830843C11DI_X05_Pin4AT %I*DI_X05_Pin_830843C11DI_X05_Pin2AT %I*DI_X05_Pin_830843C11DI_X06_Pin4AT %I*DI_X06_Pin_830843C11DI_X06_Pin2AT %I*DI_X06_Pin_830843C11DI_X07_Pin4AT %I*DI_X07_Pin_830843C11DI_X07_Pin2AT %I*DI_X07_Pin_830843C11DI_X08_Pin4AT %I*DI_X08_Pin_830843C11DI_X08_Pin2AT %I*DI_X08_Pin_830843C11DO_X01_Pin_4AT %Q*DO_X01_Pin_42CA91F71DO_X01_Pin_2AT %Q*DO_X01_Pin_42CA91F71DO_X02_Pin_4AT %Q*DO_X02_Pin_42CA91F71DO_X02_Pin_2AT %Q*DO_X02_Pin_42CA91F71DO_X03_Pin_4AT %Q*DO_X03_Pin_42CA91F71DO_X03_Pin_2AT %Q*DO_X03_Pin_42CA91F71DO_X04_Pin_4AT %Q*DO_X04_Pin_42CA91F71DO_X04_Pin_2AT %Q*DO_X04_Pin_42CA91F71DO_X05_Pin_4AT %Q*DO_X05_Pin_42CA91F71DO_X05_Pin_2AT %Q*DO_X05_Pin_42CA91F71DO_X06_Pin_4AT %Q*DO_X06_Pin_42CA91F71DO_X06_Pin_2AT %Q*DO_X06_Pin_42CA91F71DO_X07_Pin_4AT %Q*DO_X07_Pin_42CA91F71DO_X07_Pin_2AT %Q*DO_X07_Pin_42CA91F71DO_X08_Pin_4AT %Q*DO_X08_Pin_42CA91F71DO_X08_Pin_2AT %Q*DO_X08_Pin_42CA91F71WcStateAT %I*WcState_9091E0EB2InfoDataAT %I*InfoData_6F19DB2B2"}
{attribute addProperty CRC "1230247175"}
{attribute addProperty Size "36"}
TYPE EP2339_49541507 EXTENDS EtcSlaveBoxBase_77A0E4A7 :
STRUCT
	{attribute addProperty Name "DI_X01_Pin4"}
	DI_X01_Pin4 : DI_X01_Pin_830843C1;
	{attribute addProperty Name "DI_X01_Pin2"}
	DI_X01_Pin2 : DI_X01_Pin_830843C1;
	{attribute addProperty Name "DI_X02_Pin4"}
	DI_X02_Pin4 : DI_X02_Pin_830843C1;
	{attribute addProperty Name "DI_X02_Pin2"}
	DI_X02_Pin2 : DI_X02_Pin_830843C1;
	{attribute addProperty Name "DI_X03_Pin4"}
	DI_X03_Pin4 : DI_X03_Pin_830843C1;
	{attribute addProperty Name "DI_X03_Pin2"}
	DI_X03_Pin2 : DI_X03_Pin_830843C1;
	{attribute addProperty Name "DI_X04_Pin4"}
	DI_X04_Pin4 : DI_X04_Pin_830843C1;
	{attribute addProperty Name "DI_X04_Pin2"}
	DI_X04_Pin2 : DI_X04_Pin_830843C1;
	{attribute addProperty Name "DI_X05_Pin4"}
	DI_X05_Pin4 : DI_X05_Pin_830843C1;
	{attribute addProperty Name "DI_X05_Pin2"}
	DI_X05_Pin2 : DI_X05_Pin_830843C1;
	{attribute addProperty Name "DI_X06_Pin4"}
	DI_X06_Pin4 : DI_X06_Pin_830843C1;
	{attribute addProperty Name "DI_X06_Pin2"}
	DI_X06_Pin2 : DI_X06_Pin_830843C1;
	{attribute addProperty Name "DI_X07_Pin4"}
	DI_X07_Pin4 : DI_X07_Pin_830843C1;
	{attribute addProperty Name "DI_X07_Pin2"}
	DI_X07_Pin2 : DI_X07_Pin_830843C1;
	{attribute addProperty Name "DI_X08_Pin4"}
	DI_X08_Pin4 : DI_X08_Pin_830843C1;
	{attribute addProperty Name "DI_X08_Pin2"}
	DI_X08_Pin2 : DI_X08_Pin_830843C1;
	{attribute addProperty Name "DO_X01_Pin_4"}
	DO_X01_Pin_4 : DO_X01_Pin_42CA91F7;
	{attribute addProperty Name "DO_X01_Pin_2"}
	DO_X01_Pin_2 : DO_X01_Pin_42CA91F7;
	{attribute addProperty Name "DO_X02_Pin_4"}
	DO_X02_Pin_4 : DO_X02_Pin_42CA91F7;
	{attribute addProperty Name "DO_X02_Pin_2"}
	DO_X02_Pin_2 : DO_X02_Pin_42CA91F7;
	{attribute addProperty Name "DO_X03_Pin_4"}
	DO_X03_Pin_4 : DO_X03_Pin_42CA91F7;
	{attribute addProperty Name "DO_X03_Pin_2"}
	DO_X03_Pin_2 : DO_X03_Pin_42CA91F7;
	{attribute addProperty Name "DO_X04_Pin_4"}
	DO_X04_Pin_4 : DO_X04_Pin_42CA91F7;
	{attribute addProperty Name "DO_X04_Pin_2"}
	DO_X04_Pin_2 : DO_X04_Pin_42CA91F7;
	{attribute addProperty Name "DO_X05_Pin_4"}
	DO_X05_Pin_4 : DO_X05_Pin_42CA91F7;
	{attribute addProperty Name "DO_X05_Pin_2"}
	DO_X05_Pin_2 : DO_X05_Pin_42CA91F7;
	{attribute addProperty Name "DO_X06_Pin_4"}
	DO_X06_Pin_4 : DO_X06_Pin_42CA91F7;
	{attribute addProperty Name "DO_X06_Pin_2"}
	DO_X06_Pin_2 : DO_X06_Pin_42CA91F7;
	{attribute addProperty Name "DO_X07_Pin_4"}
	DO_X07_Pin_4 : DO_X07_Pin_42CA91F7;
	{attribute addProperty Name "DO_X07_Pin_2"}
	DO_X07_Pin_2 : DO_X07_Pin_42CA91F7;
	{attribute addProperty Name "DO_X08_Pin_4"}
	DO_X08_Pin_4 : DO_X08_Pin_42CA91F7;
	{attribute addProperty Name "DO_X08_Pin_2"}
	DO_X08_Pin_2 : DO_X08_Pin_42CA91F7;
	{attribute addProperty Name "WcState"}
	WcState : WcState_9091E0EB;
	{attribute addProperty Name "InfoData"}
	InfoData : InfoData_6F19DB2B;
END_STRUCT
END_TYPE

// ---- DUTs/IO/Boxes/EP2339_E3933831.TcDUT
{attribute 'GeneratedUsingTerminal: EP2339-0042-0018'}
{attribute addProperty BoxType "EP2339-0042-0018"}
{attribute addProperty Description "EP2339-0042 16 Ch. Dig. Input/Output 24V, 0.5A, M12 "}
{attribute addProperty Physics "YY"}
{attribute addProperty Id "DI_X01_4AT %I*DI_X_830843C11DI_X01_2AT %I*DI_X_830843C11DI_X02_4AT %I*DI_X_830843C11DI_X02_2AT %I*DI_X_830843C11DI_X03_4AT %I*DI_X_830843C11DI_X03_2AT %I*DI_X_830843C11DI_X04_4AT %I*DI_X_830843C11DI_X04_2AT %I*DI_X_830843C11DI_X05_4AT %I*DI_X_830843C11DI_X05_2AT %I*DI_X_830843C11DI_X06_4AT %I*DI_X_830843C11DI_X06_2AT %I*DI_X_830843C11DI_X07_4AT %I*DI_X_830843C11DI_X07_2AT %I*DI_X_830843C11DI_X08_4AT %I*DI_X_830843C11DI_X08_2AT %I*DI_X_830843C11DO_X01_4AT %Q*DO_X_42CA91F71DO_X01_2AT %Q*DO_X_42CA91F71DO_X02_4AT %Q*DO_X_42CA91F71DO_X02_2AT %Q*DO_X_42CA91F71DO_X03_4AT %Q*DO_X_42CA91F71DO_X03_2AT %Q*DO_X_42CA91F71DO_X04_4AT %Q*DO_X_42CA91F71DO_X04_2AT %Q*DO_X_42CA91F71DO_X05_4AT %Q*DO_X_42CA91F71DO_X05_2AT %Q*DO_X_42CA91F71DO_X06_4AT %Q*DO_X_42CA91F71DO_X06_2AT %Q*DO_X_42CA91F71DO_X07_4AT %Q*DO_X_42CA91F71DO_X07_2AT %Q*DO_X_42CA91F71DO_X08_4AT %Q*DO_X_42CA91F71DO_X08_2AT %Q*DO_X_42CA91F71WcStateAT %I*WcState_9091E0EB2InfoDataAT %I*InfoData_6F19DB2B2"}
{attribute addProperty CRC "3818076209"}
{attribute addProperty Size "36"}
TYPE EP2339_E3933831 EXTENDS EtcSlaveBoxBase_77A0E4A7 :
STRUCT
	{attribute addProperty Name "DI_X01_4"}
	DI_X01_4 : DI_X_830843C1;
	{attribute addProperty Name "DI_X01_2"}
	DI_X01_2 : DI_X_830843C1;
	{attribute addProperty Name "DI_X02_4"}
	DI_X02_4 : DI_X_830843C1;
	{attribute addProperty Name "DI_X02_2"}
	DI_X02_2 : DI_X_830843C1;
	{attribute addProperty Name "DI_X03_4"}
	DI_X03_4 : DI_X_830843C1;
	{attribute addProperty Name "DI_X03_2"}
	DI_X03_2 : DI_X_830843C1;
	{attribute addProperty Name "DI_X04_4"}
	DI_X04_4 : DI_X_830843C1;
	{attribute addProperty Name "DI_X04_2"}
	DI_X04_2 : DI_X_830843C1;
	{attribute addProperty Name "DI_X05_4"}
	DI_X05_4 : DI_X_830843C1;
	{attribute addProperty Name "DI_X05_2"}
	DI_X05_2 : DI_X_830843C1;
	{attribute addProperty Name "DI_X06_4"}
	DI_X06_4 : DI_X_830843C1;
	{attribute addProperty Name "DI_X06_2"}
	DI_X06_2 : DI_X_830843C1;
	{attribute addProperty Name "DI_X07_4"}
	DI_X07_4 : DI_X_830843C1;
	{attribute addProperty Name "DI_X07_2"}
	DI_X07_2 : DI_X_830843C1;
	{attribute addProperty Name "DI_X08_4"}
	DI_X08_4 : DI_X_830843C1;
	{attribute addProperty Name "DI_X08_2"}
	DI_X08_2 : DI_X_830843C1;
	{attribute addProperty Name "DO_X01_4"}
	DO_X01_4 : DO_X_42CA91F7;
	{attribute addProperty Name "DO_X01_2"}
	DO_X01_2 : DO_X_42CA91F7;
	{attribute addProperty Name "DO_X02_4"}
	DO_X02_4 : DO_X_42CA91F7;
	{attribute addProperty Name "DO_X02_2"}
	DO_X02_2 : DO_X_42CA91F7;
	{attribute addProperty Name "DO_X03_4"}
	DO_X03_4 : DO_X_42CA91F7;
	{attribute addProperty Name "DO_X03_2"}
	DO_X03_2 : DO_X_42CA91F7;
	{attribute addProperty Name "DO_X04_4"}
	DO_X04_4 : DO_X_42CA91F7;
	{attribute addProperty Name "DO_X04_2"}
	DO_X04_2 : DO_X_42CA91F7;
	{attribute addProperty Name "DO_X05_4"}
	DO_X05_4 : DO_X_42CA91F7;
	{attribute addProperty Name "DO_X05_2"}
	DO_X05_2 : DO_X_42CA91F7;
	{attribute addProperty Name "DO_X06_4"}
	DO_X06_4 : DO_X_42CA91F7;
	{attribute addProperty Name "DO_X06_2"}
	DO_X06_2 : DO_X_42CA91F7;
	{attribute addProperty Name "DO_X07_4"}
	DO_X07_4 : DO_X_42CA91F7;
	{attribute addProperty Name "DO_X07_2"}
	DO_X07_2 : DO_X_42CA91F7;
	{attribute addProperty Name "DO_X08_4"}
	DO_X08_4 : DO_X_42CA91F7;
	{attribute addProperty Name "DO_X08_2"}
	DO_X08_2 : DO_X_42CA91F7;
	{attribute addProperty Name "WcState"}
	WcState : WcState_9091E0EB;
	{attribute addProperty Name "InfoData"}
	InfoData : InfoData_6F19DB2B;
END_STRUCT
END_TYPE

// ---- DUTs/IO/Boxes/EP2349_4CF33DED.TcDUT
{attribute 'GeneratedUsingTerminal: EP2349-0021-0016'}
{attribute addProperty BoxType "EP2349-0021-0016"}
{attribute addProperty Description "EP2349-0021 16 Ch. Dig. Input/Output 24V, 10µs, 0,5A, M8"}
{attribute addProperty Physics "YY"}
{attribute addProperty Id "Channel_1AT %I*Channel_830843C11Channel_2AT %I*Channel_830843C11Channel_3AT %I*Channel_830843C11Channel_4AT %I*Channel_830843C11Channel_5AT %I*Channel_830843C11Channel_6AT %I*Channel_830843C11Channel_7AT %I*Channel_830843C11Channel_8AT %I*Channel_830843C11Channel_9AT %I*Channel_830843C11Channel_10AT %I*Channel_830843C11Channel_11AT %I*Channel_830843C11Channel_12AT %I*Channel_830843C11Channel_13AT %I*Channel_830843C11Channel_14AT %I*Channel_830843C11Channel_15AT %I*Channel_830843C11Channel_16AT %I*Channel_830843C11Channel_17AT %Q*Channel_42CA91F71Channel_18AT %Q*Channel_42CA91F71Channel_19AT %Q*Channel_42CA91F71Channel_20AT %Q*Channel_42CA91F71Channel_21AT %Q*Channel_42CA91F71Channel_22AT %Q*Channel_42CA91F71Channel_23AT %Q*Channel_42CA91F71Channel_24AT %Q*Channel_42CA91F71Channel_25AT %Q*Channel_42CA91F71Channel_26AT %Q*Channel_42CA91F71Channel_27AT %Q*Channel_42CA91F71Channel_28AT %Q*Channel_42CA91F71Channel_29AT %Q*Channel_42CA91F71Channel_30AT %Q*Channel_42CA91F71Channel_31AT %Q*Channel_42CA91F71Channel_32AT %Q*Channel_42CA91F71WcStateAT %I*WcState_9091E0EB2InfoDataAT %I*InfoData_6F19DB2B2"}
{attribute addProperty CRC "1291009517"}
{attribute addProperty Size "36"}
TYPE EP2349_4CF33DED EXTENDS EtcSlaveBoxBase_77A0E4A7 :
STRUCT
	{attribute addProperty Name "Channel_1"}
	Channel_1 : Channel_830843C1;
	{attribute addProperty Name "Channel_2"}
	Channel_2 : Channel_830843C1;
	{attribute addProperty Name "Channel_3"}
	Channel_3 : Channel_830843C1;
	{attribute addProperty Name "Channel_4"}
	Channel_4 : Channel_830843C1;
	{attribute addProperty Name "Channel_5"}
	Channel_5 : Channel_830843C1;
	{attribute addProperty Name "Channel_6"}
	Channel_6 : Channel_830843C1;
	{attribute addProperty Name "Channel_7"}
	Channel_7 : Channel_830843C1;
	{attribute addProperty Name "Channel_8"}
	Channel_8 : Channel_830843C1;
	{attribute addProperty Name "Channel_9"}
	Channel_9 : Channel_830843C1;
	{attribute addProperty Name "Channel_10"}
	Channel_10 : Channel_830843C1;
	{attribute addProperty Name "Channel_11"}
	Channel_11 : Channel_830843C1;
	{attribute addProperty Name "Channel_12"}
	Channel_12 : Channel_830843C1;
	{attribute addProperty Name "Channel_13"}
	Channel_13 : Channel_830843C1;
	{attribute addProperty Name "Channel_14"}
	Channel_14 : Channel_830843C1;
	{attribute addProperty Name "Channel_15"}
	Channel_15 : Channel_830843C1;
	{attribute addProperty Name "Channel_16"}
	Channel_16 : Channel_830843C1;
	{attribute addProperty Name "Channel_17"}
	Channel_17 : Channel_42CA91F7;
	{attribute addProperty Name "Channel_18"}
	Channel_18 : Channel_42CA91F7;
	{attribute addProperty Name "Channel_19"}
	Channel_19 : Channel_42CA91F7;
	{attribute addProperty Name "Channel_20"}
	Channel_20 : Channel_42CA91F7;
	{attribute addProperty Name "Channel_21"}
	Channel_21 : Channel_42CA91F7;
	{attribute addProperty Name "Channel_22"}
	Channel_22 : Channel_42CA91F7;
	{attribute addProperty Name "Channel_23"}
	Channel_23 : Channel_42CA91F7;
	{attribute addProperty Name "Channel_24"}
	Channel_24 : Channel_42CA91F7;
	{attribute addProperty Name "Channel_25"}
	Channel_25 : Channel_42CA91F7;
	{attribute addProperty Name "Channel_26"}
	Channel_26 : Channel_42CA91F7;
	{attribute addProperty Name "Channel_27"}
	Channel_27 : Channel_42CA91F7;
	{attribute addProperty Name "Channel_28"}
	Channel_28 : Channel_42CA91F7;
	{attribute addProperty Name "Channel_29"}
	Channel_29 : Channel_42CA91F7;
	{attribute addProperty Name "Channel_30"}
	Channel_30 : Channel_42CA91F7;
	{attribute addProperty Name "Channel_31"}
	Channel_31 : Channel_42CA91F7;
	{attribute addProperty Name "Channel_32"}
	Channel_32 : Channel_42CA91F7;
	{attribute addProperty Name "WcState"}
	WcState : WcState_9091E0EB;
	{attribute addProperty Name "InfoData"}
	InfoData : InfoData_6F19DB2B;
END_STRUCT
END_TYPE

// ---- DUTs/IO/Boxes/EP2624_7B64371E.TcDUT
{attribute 'GeneratedUsingTerminal: EP2624-0002-0016'}
{attribute addProperty BoxType "EP2624-0002-0016"}
{attribute addProperty Description "EP2624-0002 4Ch. Relay Output, NO (125V AC / 30V DC)"}
{attribute addProperty Physics "YY"}
{attribute addProperty Id "Channel_1AT %Q*Channel_42CA91F71Channel_2AT %Q*Channel_42CA91F71Channel_3AT %Q*Channel_42CA91F71Channel_4AT %Q*Channel_42CA91F71WcStateAT %I*WcState_0B2B16F91InfoDataAT %I*InfoData_6F19DB2B2"}
{attribute addProperty CRC "2070165278"}
{attribute addProperty Size "7"}
TYPE EP2624_7B64371E EXTENDS EtcSlaveBoxBase_77A0E4A7 :
STRUCT
	{attribute addProperty Name "Channel_1"}
	Channel_1 : Channel_42CA91F7;
	{attribute addProperty Name "Channel_2"}
	Channel_2 : Channel_42CA91F7;
	{attribute addProperty Name "Channel_3"}
	Channel_3 : Channel_42CA91F7;
	{attribute addProperty Name "Channel_4"}
	Channel_4 : Channel_42CA91F7;
	{attribute addProperty Name "WcState"}
	WcState : WcState_0B2B16F9;
	{attribute addProperty Name "InfoData"}
	InfoData : InfoData_6F19DB2B;
END_STRUCT
END_TYPE

// ---- DUTs/IO/Boxes/EP2809_2B6483BD.TcDUT
{attribute 'GeneratedUsingTerminal: EP2809-0021-0016'}
{attribute addProperty BoxType "EP2809-0021-0016"}
{attribute addProperty Description "EP2809-0021 16 Ch. Dig. Output 24V, 0,5A, M8"}
{attribute addProperty Physics "YY"}
{attribute addProperty Id "Channel_1AT %Q*Channel_42CA91F71Channel_2AT %Q*Channel_42CA91F71Channel_3AT %Q*Channel_42CA91F71Channel_4AT %Q*Channel_42CA91F71Channel_5AT %Q*Channel_42CA91F71Channel_6AT %Q*Channel_42CA91F71Channel_7AT %Q*Channel_42CA91F71Channel_8AT %Q*Channel_42CA91F71Channel_9AT %Q*Channel_42CA91F71Channel_10AT %Q*Channel_42CA91F71Channel_11AT %Q*Channel_42CA91F71Channel_12AT %Q*Channel_42CA91F71Channel_13AT %Q*Channel_42CA91F71Channel_14AT %Q*Channel_42CA91F71Channel_15AT %Q*Channel_42CA91F71Channel_16AT %Q*Channel_42CA91F71WcStateAT %I*WcState_0B2B16F91InfoDataAT %I*InfoData_6F19DB2B2"}
{attribute addProperty CRC "728007613"}
{attribute addProperty Size "19"}
TYPE EP2809_2B6483BD EXTENDS EtcSlaveBoxBase_77A0E4A7 :
STRUCT
	{attribute addProperty Name "Channel_1"}
	Channel_1 : Channel_42CA91F7;
	{attribute addProperty Name "Channel_2"}
	Channel_2 : Channel_42CA91F7;
	{attribute addProperty Name "Channel_3"}
	Channel_3 : Channel_42CA91F7;
	{attribute addProperty Name "Channel_4"}
	Channel_4 : Channel_42CA91F7;
	{attribute addProperty Name "Channel_5"}
	Channel_5 : Channel_42CA91F7;
	{attribute addProperty Name "Channel_6"}
	Channel_6 : Channel_42CA91F7;
	{attribute addProperty Name "Channel_7"}
	Channel_7 : Channel_42CA91F7;
	{attribute addProperty Name "Channel_8"}
	Channel_8 : Channel_42CA91F7;
	{attribute addProperty Name "Channel_9"}
	Channel_9 : Channel_42CA91F7;
	{attribute addProperty Name "Channel_10"}
	Channel_10 : Channel_42CA91F7;
	{attribute addProperty Name "Channel_11"}
	Channel_11 : Channel_42CA91F7;
	{attribute addProperty Name "Channel_12"}
	Channel_12 : Channel_42CA91F7;
	{attribute addProperty Name "Channel_13"}
	Channel_13 : Channel_42CA91F7;
	{attribute addProperty Name "Channel_14"}
	Channel_14 : Channel_42CA91F7;
	{attribute addProperty Name "Channel_15"}
	Channel_15 : Channel_42CA91F7;
	{attribute addProperty Name "Channel_16"}
	Channel_16 : Channel_42CA91F7;
	{attribute addProperty Name "WcState"}
	WcState : WcState_0B2B16F9;
	{attribute addProperty Name "InfoData"}
	InfoData : InfoData_6F19DB2B;
END_STRUCT
END_TYPE

// ---- DUTs/IO/Boxes/EP2809_7AAF2E71.TcDUT
{attribute 'GeneratedUsingTerminal: EP2809-0042-0017'}
{attribute addProperty BoxType "EP2809-0042-0017"}
{attribute addProperty Description "EP2809-0042 16 Ch. Dig. Output 24V, 0,5A, M12"}
{attribute addProperty Physics "YY"}
{attribute addProperty Id "DO_X01_Pin_4AT %Q*DO_X01_Pin_42CA91F71DO_X01_Pin_2AT %Q*DO_X01_Pin_42CA91F71DO_X02_Pin_4AT %Q*DO_X02_Pin_42CA91F71DO_X02_Pin_2AT %Q*DO_X02_Pin_42CA91F71DO_X03_Pin_4AT %Q*DO_X03_Pin_42CA91F71DO_X03_Pin_2AT %Q*DO_X03_Pin_42CA91F71DO_X04_Pin_4AT %Q*DO_X04_Pin_42CA91F71DO_X04_Pin_2AT %Q*DO_X04_Pin_42CA91F71DO_X05_Pin_4AT %Q*DO_X05_Pin_42CA91F71DO_X05_Pin_2AT %Q*DO_X05_Pin_42CA91F71DO_X06_Pin_4AT %Q*DO_X06_Pin_42CA91F71DO_X06_Pin_2AT %Q*DO_X06_Pin_42CA91F71DO_X07_Pin_4AT %Q*DO_X07_Pin_42CA91F71DO_X07_Pin_2AT %Q*DO_X07_Pin_42CA91F71DO_X08_Pin_4AT %Q*DO_X08_Pin_42CA91F71DO_X08_Pin_2AT %Q*DO_X08_Pin_42CA91F71WcStateAT %I*WcState_0B2B16F91InfoDataAT %I*InfoData_6F19DB2B2"}
{attribute addProperty CRC "2058301041"}
{attribute addProperty Size "19"}
TYPE EP2809_7AAF2E71 EXTENDS EtcSlaveBoxBase_77A0E4A7 :
STRUCT
	{attribute addProperty Name "DO_X01_Pin_4"}
	DO_X01_Pin_4 : DO_X01_Pin_42CA91F7;
	{attribute addProperty Name "DO_X01_Pin_2"}
	DO_X01_Pin_2 : DO_X01_Pin_42CA91F7;
	{attribute addProperty Name "DO_X02_Pin_4"}
	DO_X02_Pin_4 : DO_X02_Pin_42CA91F7;
	{attribute addProperty Name "DO_X02_Pin_2"}
	DO_X02_Pin_2 : DO_X02_Pin_42CA91F7;
	{attribute addProperty Name "DO_X03_Pin_4"}
	DO_X03_Pin_4 : DO_X03_Pin_42CA91F7;
	{attribute addProperty Name "DO_X03_Pin_2"}
	DO_X03_Pin_2 : DO_X03_Pin_42CA91F7;
	{attribute addProperty Name "DO_X04_Pin_4"}
	DO_X04_Pin_4 : DO_X04_Pin_42CA91F7;
	{attribute addProperty Name "DO_X04_Pin_2"}
	DO_X04_Pin_2 : DO_X04_Pin_42CA91F7;
	{attribute addProperty Name "DO_X05_Pin_4"}
	DO_X05_Pin_4 : DO_X05_Pin_42CA91F7;
	{attribute addProperty Name "DO_X05_Pin_2"}
	DO_X05_Pin_2 : DO_X05_Pin_42CA91F7;
	{attribute addProperty Name "DO_X06_Pin_4"}
	DO_X06_Pin_4 : DO_X06_Pin_42CA91F7;
	{attribute addProperty Name "DO_X06_Pin_2"}
	DO_X06_Pin_2 : DO_X06_Pin_42CA91F7;
	{attribute addProperty Name "DO_X07_Pin_4"}
	DO_X07_Pin_4 : DO_X07_Pin_42CA91F7;
	{attribute addProperty Name "DO_X07_Pin_2"}
	DO_X07_Pin_2 : DO_X07_Pin_42CA91F7;
	{attribute addProperty Name "DO_X08_Pin_4"}
	DO_X08_Pin_4 : DO_X08_Pin_42CA91F7;
	{attribute addProperty Name "DO_X08_Pin_2"}
	DO_X08_Pin_2 : DO_X08_Pin_42CA91F7;
	{attribute addProperty Name "WcState"}
	WcState : WcState_0B2B16F9;
	{attribute addProperty Name "InfoData"}
	InfoData : InfoData_6F19DB2B;
END_STRUCT
END_TYPE

// ---- DUTs/IO/Boxes/EP2809_23623E9C.TcDUT
{attribute 'GeneratedUsingTerminal: EP2809-0042-0018'}
{attribute addProperty BoxType "EP2809-0042-0018"}
{attribute addProperty Description "EP2809-0042 16 Ch. Dig. Output 24V, 0,5A, M12"}
{attribute addProperty Physics "YY"}
{attribute addProperty Id "DO_X01_4AT %Q*DO_X_42CA91F71DO_X01_2AT %Q*DO_X_42CA91F71DO_X02_4AT %Q*DO_X_42CA91F71DO_X02_2AT %Q*DO_X_42CA91F71DO_X03_4AT %Q*DO_X_42CA91F71DO_X03_2AT %Q*DO_X_42CA91F71DO_X04_4AT %Q*DO_X_42CA91F71DO_X04_2AT %Q*DO_X_42CA91F71DO_X05_4AT %Q*DO_X_42CA91F71DO_X05_2AT %Q*DO_X_42CA91F71DO_X06_4AT %Q*DO_X_42CA91F71DO_X06_2AT %Q*DO_X_42CA91F71DO_X07_4AT %Q*DO_X_42CA91F71DO_X07_2AT %Q*DO_X_42CA91F71DO_X08_4AT %Q*DO_X_42CA91F71DO_X08_2AT %Q*DO_X_42CA91F71WcStateAT %I*WcState_0B2B16F91InfoDataAT %I*InfoData_6F19DB2B2"}
{attribute addProperty CRC "593641116"}
{attribute addProperty Size "19"}
TYPE EP2809_23623E9C EXTENDS EtcSlaveBoxBase_77A0E4A7 :
STRUCT
	{attribute addProperty Name "DO_X01_4"}
	DO_X01_4 : DO_X_42CA91F7;
	{attribute addProperty Name "DO_X01_2"}
	DO_X01_2 : DO_X_42CA91F7;
	{attribute addProperty Name "DO_X02_4"}
	DO_X02_4 : DO_X_42CA91F7;
	{attribute addProperty Name "DO_X02_2"}
	DO_X02_2 : DO_X_42CA91F7;
	{attribute addProperty Name "DO_X03_4"}
	DO_X03_4 : DO_X_42CA91F7;
	{attribute addProperty Name "DO_X03_2"}
	DO_X03_2 : DO_X_42CA91F7;
	{attribute addProperty Name "DO_X04_4"}
	DO_X04_4 : DO_X_42CA91F7;
	{attribute addProperty Name "DO_X04_2"}
	DO_X04_2 : DO_X_42CA91F7;
	{attribute addProperty Name "DO_X05_4"}
	DO_X05_4 : DO_X_42CA91F7;
	{attribute addProperty Name "DO_X05_2"}
	DO_X05_2 : DO_X_42CA91F7;
	{attribute addProperty Name "DO_X06_4"}
	DO_X06_4 : DO_X_42CA91F7;
	{attribute addProperty Name "DO_X06_2"}
	DO_X06_2 : DO_X_42CA91F7;
	{attribute addProperty Name "DO_X07_4"}
	DO_X07_4 : DO_X_42CA91F7;
	{attribute addProperty Name "DO_X07_2"}
	DO_X07_2 : DO_X_42CA91F7;
	{attribute addProperty Name "DO_X08_4"}
	DO_X08_4 : DO_X_42CA91F7;
	{attribute addProperty Name "DO_X08_2"}
	DO_X08_2 : DO_X_42CA91F7;
	{attribute addProperty Name "WcState"}
	WcState : WcState_0B2B16F9;
	{attribute addProperty Name "InfoData"}
	InfoData : InfoData_6F19DB2B;
END_STRUCT
END_TYPE

// ---- DUTs/IO/Boxes/EP2816_F9F6AB82.TcDUT
{attribute 'GeneratedUsingTerminal: EP2816-0003-0016'}
{attribute addProperty BoxType "EP2816-0003-0016"}
{attribute addProperty Description "EP2816-0003 16CH. Dig. Output, Diagnostic, 10-Pole Plug Connector"}
{attribute addProperty Physics "YY"}
{attribute addProperty Id "DIG_Diag_Inputs_Channel_1AT %I*DIG_Diag_Inputs_Channel_584303BF8DIG_Diag_Inputs_Channel_2AT %I*DIG_Diag_Inputs_Channel_584303BF8DIG_Inputs_DeviceAT %I*DIG_Inputs_Device_E94E5BF95DIG_Output_Channel_1AT %Q*DIG_Output_Channel_28AC1A9E8DIG_Output_Channel_2AT %Q*DIG_Output_Channel_28AC1A9E8DIG_Outputs_DeviceAT %Q*DIG_Outputs_Device_36A5EF172WcStateAT %I*WcState_9091E0EB2InfoDataAT %I*InfoData_32EB74EA10"}
{attribute addProperty CRC "4193692546"}
{attribute addProperty Size "51"}
TYPE EP2816_F9F6AB82 EXTENDS EtcSlaveBoxBase_77A0E4A7 :
STRUCT
	{attribute addProperty Name "DIG_Diag_Inputs_Channel_1"}
	DIG_Diag_Inputs_Channel_1 : DIG_Diag_Inputs_Channel_584303BF;
	{attribute addProperty Name "DIG_Diag_Inputs_Channel_2"}
	DIG_Diag_Inputs_Channel_2 : DIG_Diag_Inputs_Channel_584303BF;
	{attribute addProperty Name "DIG_Inputs_Device"}
	DIG_Inputs_Device : DIG_Inputs_Device_E94E5BF9;
	{attribute addProperty Name "DIG_Output_Channel_1"}
	DIG_Output_Channel_1 : DIG_Output_Channel_28AC1A9E;
	{attribute addProperty Name "DIG_Output_Channel_2"}
	DIG_Output_Channel_2 : DIG_Output_Channel_28AC1A9E;
	{attribute addProperty Name "DIG_Outputs_Device"}
	DIG_Outputs_Device : DIG_Outputs_Device_36A5EF17;
	{attribute addProperty Name "WcState"}
	WcState : WcState_9091E0EB;
	{attribute addProperty Name "InfoData"}
	InfoData : InfoData_32EB74EA;
END_STRUCT
END_TYPE

// ---- DUTs/IO/Boxes/EP2816_88324133.TcDUT
{attribute 'GeneratedUsingTerminal: EP2816-0004-0016'}
{attribute addProperty BoxType "EP2816-0004-0016"}
{attribute addProperty Description "EP2816-0004 16 Ch. Dig. Output 24V, 0,5A, M16"}
{attribute addProperty Physics "YY"}
{attribute addProperty Id "DO_Outputs_Channel_1AT %Q*DO_Outputs_Channel_28AC1A9E8DO_Outputs_Channel_2AT %Q*DO_Outputs_Channel_28AC1A9E8WcStateAT %I*WcState_0B2B16F91InfoDataAT %I*InfoData_32EB74EA10"}
{attribute addProperty CRC "2284994867"}
{attribute addProperty Size "27"}
TYPE EP2816_88324133 EXTENDS EtcSlaveBoxBase_77A0E4A7 :
STRUCT
	{attribute addProperty Name "DO_Outputs_Channel_1"}
	DO_Outputs_Channel_1 : DO_Outputs_Channel_28AC1A9E;
	{attribute addProperty Name "DO_Outputs_Channel_2"}
	DO_Outputs_Channel_2 : DO_Outputs_Channel_28AC1A9E;
	{attribute addProperty Name "WcState"}
	WcState : WcState_0B2B16F9;
	{attribute addProperty Name "InfoData"}
	InfoData : InfoData_32EB74EA;
END_STRUCT
END_TYPE

// ---- DUTs/IO/Boxes/EP2816_0C961E28.TcDUT
{attribute 'GeneratedUsingTerminal: EP2816-0008-0016'}
{attribute addProperty BoxType "EP2816-0008-0016"}
{attribute addProperty Description "EP2816-0008 16 Ch. Dig. Output 24V, 0,5A, Diagnostic, D-SUB25"}
{attribute addProperty Physics "YY"}
{attribute addProperty Id "DO_Inputs_Channel_1AT %I*DO_Inputs_Channel_584303BF8DO_Inputs_Channel_2AT %I*DO_Inputs_Channel_584303BF8DO_Inputs_DeviceAT %I*DO_Inputs_Device_4E5AF17E5DO_Outputs_Channel_1AT %Q*DO_Outputs_Channel_28AC1A9E8DO_Outputs_Channel_2AT %Q*DO_Outputs_Channel_28AC1A9E8DO_Outputs_DeviceAT %Q*DO_Outputs_Device_36A5EF172WcStateAT %I*WcState_9091E0EB2InfoDataAT %I*InfoData_32EB74EA10"}
{attribute addProperty CRC "211164712"}
{attribute addProperty Size "51"}
TYPE EP2816_0C961E28 EXTENDS EtcSlaveBoxBase_77A0E4A7 :
STRUCT
	{attribute addProperty Name "DO_Inputs_Channel_1"}
	DO_Inputs_Channel_1 : DO_Inputs_Channel_584303BF;
	{attribute addProperty Name "DO_Inputs_Channel_2"}
	DO_Inputs_Channel_2 : DO_Inputs_Channel_584303BF;
	{attribute addProperty Name "DO_Inputs_Device"}
	DO_Inputs_Device : DO_Inputs_Device_4E5AF17E;
	{attribute addProperty Name "DO_Outputs_Channel_1"}
	DO_Outputs_Channel_1 : DO_Outputs_Channel_28AC1A9E;
	{attribute addProperty Name "DO_Outputs_Channel_2"}
	DO_Outputs_Channel_2 : DO_Outputs_Channel_28AC1A9E;
	{attribute addProperty Name "DO_Outputs_Device"}
	DO_Outputs_Device : DO_Outputs_Device_36A5EF17;
	{attribute addProperty Name "WcState"}
	WcState : WcState_9091E0EB;
	{attribute addProperty Name "InfoData"}
	InfoData : InfoData_32EB74EA;
END_STRUCT
END_TYPE

// ---- DUTs/IO/Boxes/EP2816_D9B77CAE.TcDUT
{attribute 'GeneratedUsingTerminal: EP2816-0008-0018'}
{attribute addProperty BoxType "EP2816-0008-0018"}
{attribute addProperty Description "EP2816-0008 16 Ch. Dig. Output 24V, 0,5A, Diagnostic, D-SUB25"}
{attribute addProperty Physics "YY"}
{attribute addProperty Id "DIG_Diag_Inputs_Channel_1AT %I*DIG_Diag_Inputs_Channel_584303BF8DIG_Diag_Inputs_Channel_2AT %I*DIG_Diag_Inputs_Channel_584303BF8DIG_Inputs_DeviceAT %I*DIG_Inputs_Device_4E5AF17E5DIG_Outputs_Channel_1AT %Q*DIG_Outputs_Channel_28AC1A9E8DIG_Outputs_Channel_2AT %Q*DIG_Outputs_Channel_28AC1A9E8DIG_Outputs_DeviceAT %Q*DIG_Outputs_Device_36A5EF172WcStateAT %I*WcState_9091E0EB2InfoDataAT %I*InfoData_32EB74EA10"}
{attribute addProperty CRC "3652680878"}
{attribute addProperty Size "51"}
TYPE EP2816_D9B77CAE EXTENDS EtcSlaveBoxBase_77A0E4A7 :
STRUCT
	{attribute addProperty Name "DIG_Diag_Inputs_Channel_1"}
	DIG_Diag_Inputs_Channel_1 : DIG_Diag_Inputs_Channel_584303BF;
	{attribute addProperty Name "DIG_Diag_Inputs_Channel_2"}
	DIG_Diag_Inputs_Channel_2 : DIG_Diag_Inputs_Channel_584303BF;
	{attribute addProperty Name "DIG_Inputs_Device"}
	DIG_Inputs_Device : DIG_Inputs_Device_4E5AF17E;
	{attribute addProperty Name "DIG_Outputs_Channel_1"}
	DIG_Outputs_Channel_1 : DIG_Outputs_Channel_28AC1A9E;
	{attribute addProperty Name "DIG_Outputs_Channel_2"}
	DIG_Outputs_Channel_2 : DIG_Outputs_Channel_28AC1A9E;
	{attribute addProperty Name "DIG_Outputs_Device"}
	DIG_Outputs_Device : DIG_Outputs_Device_36A5EF17;
	{attribute addProperty Name "WcState"}
	WcState : WcState_9091E0EB;
	{attribute addProperty Name "InfoData"}
	InfoData : InfoData_32EB74EA;
END_STRUCT
END_TYPE

// ---- DUTs/IO/Boxes/EP2816_01296449.TcDUT
{attribute 'GeneratedUsingTerminal: EP2816-0008-0019'}
{attribute addProperty BoxType "EP2816-0008-0019"}
{attribute addProperty Description "EP2816-0008 16 Ch. Dig. Output 24V, 0,5A, Diagnostic, D-SUB25"}
{attribute addProperty Physics "YY"}
{attribute addProperty Id "DIG_Diag_Inputs_Channel_1AT %I*DIG_Diag_Inputs_Channel_584303BF8DIG_Diag_Inputs_Channel_2AT %I*DIG_Diag_Inputs_Channel_584303BF8DIG_Inputs_DeviceAT %I*DIG_Inputs_Device_E94E5BF95DIG_Outputs_Channel_1AT %Q*DIG_Outputs_Channel_28AC1A9E8DIG_Outputs_Channel_2AT %Q*DIG_Outputs_Channel_28AC1A9E8DIG_Outputs_DeviceAT %Q*DIG_Outputs_Device_36A5EF172WcStateAT %I*WcState_9091E0EB2InfoDataAT %I*InfoData_32EB74EA10"}
{attribute addProperty CRC "19489865"}
{attribute addProperty Size "51"}
TYPE EP2816_01296449 EXTENDS EtcSlaveBoxBase_77A0E4A7 :
STRUCT
	{attribute addProperty Name "DIG_Diag_Inputs_Channel_1"}
	DIG_Diag_Inputs_Channel_1 : DIG_Diag_Inputs_Channel_584303BF;
	{attribute addProperty Name "DIG_Diag_Inputs_Channel_2"}
	DIG_Diag_Inputs_Channel_2 : DIG_Diag_Inputs_Channel_584303BF;
	{attribute addProperty Name "DIG_Inputs_Device"}
	DIG_Inputs_Device : DIG_Inputs_Device_E94E5BF9;
	{attribute addProperty Name "DIG_Outputs_Channel_1"}
	DIG_Outputs_Channel_1 : DIG_Outputs_Channel_28AC1A9E;
	{attribute addProperty Name "DIG_Outputs_Channel_2"}
	DIG_Outputs_Channel_2 : DIG_Outputs_Channel_28AC1A9E;
	{attribute addProperty Name "DIG_Outputs_Device"}
	DIG_Outputs_Device : DIG_Outputs_Device_36A5EF17;
	{attribute addProperty Name "WcState"}
	WcState : WcState_9091E0EB;
	{attribute addProperty Name "InfoData"}
	InfoData : InfoData_32EB74EA;
END_STRUCT
END_TYPE

// ---- DUTs/IO/Boxes/EP2817_7CB3CE29.TcDUT
{attribute 'GeneratedUsingTerminal: EP2817-0008-0016'}
{attribute addProperty BoxType "EP2817-0008-0016"}
{attribute addProperty Description "EP2817-0008 24Ch. Dig. Output 24V 0,5A, Diagnostics, D-SUB25"}
{attribute addProperty Physics "YY"}
{attribute addProperty Id "DIG_Diag_Inputs_Channel_1AT %I*DIG_Diag_Inputs_Channel_584303BF8DIG_Diag_Inputs_Channel_2AT %I*DIG_Diag_Inputs_Channel_584303BF8DIG_Diag_Inputs_Channel_3AT %I*DIG_Diag_Inputs_Channel_584303BF8DIG_Inputs_DeviceAT %I*DIG_Inputs_Device_27CCC8668DIG_Output_Channel_1AT %Q*DIG_Output_Channel_28AC1A9E8DIG_Output_Channel_2AT %Q*DIG_Output_Channel_28AC1A9E8DIG_Output_Channel_3AT %Q*DIG_Output_Channel_28AC1A9E8DIG_Outputs_DeviceAT %Q*DIG_Outputs_Device_36A5EF172WcStateAT %I*WcState_9091E0EB2InfoDataAT %I*InfoData_32EB74EA10"}
{attribute addProperty CRC "2092158505"}
{attribute addProperty Size "70"}
TYPE EP2817_7CB3CE29 EXTENDS EtcSlaveBoxBase_77A0E4A7 :
STRUCT
	{attribute addProperty Name "DIG_Diag_Inputs_Channel_1"}
	DIG_Diag_Inputs_Channel_1 : DIG_Diag_Inputs_Channel_584303BF;
	{attribute addProperty Name "DIG_Diag_Inputs_Channel_2"}
	DIG_Diag_Inputs_Channel_2 : DIG_Diag_Inputs_Channel_584303BF;
	{attribute addProperty Name "DIG_Diag_Inputs_Channel_3"}
	DIG_Diag_Inputs_Channel_3 : DIG_Diag_Inputs_Channel_584303BF;
	{attribute addProperty Name "DIG_Inputs_Device"}
	DIG_Inputs_Device : DIG_Inputs_Device_27CCC866;
	{attribute addProperty Name "DIG_Output_Channel_1"}
	DIG_Output_Channel_1 : DIG_Output_Channel_28AC1A9E;
	{attribute addProperty Name "DIG_Output_Channel_2"}
	DIG_Output_Channel_2 : DIG_Output_Channel_28AC1A9E;
	{attribute addProperty Name "DIG_Output_Channel_3"}
	DIG_Output_Channel_3 : DIG_Output_Channel_28AC1A9E;
	{attribute addProperty Name "DIG_Outputs_Device"}
	DIG_Outputs_Device : DIG_Outputs_Device_36A5EF17;
	{attribute addProperty Name "WcState"}
	WcState : WcState_9091E0EB;
	{attribute addProperty Name "InfoData"}
	InfoData : InfoData_32EB74EA;
END_STRUCT
END_TYPE

// ---- DUTs/IO/Boxes/EP3162_AA20D87B.TcDUT
{attribute 'GeneratedUsingTerminal: EP3162-0002-0016'}
{attribute addProperty BoxType "EP3162-0002-0016"}
{attribute addProperty Description "EP3162-0002 2Ch. Ana. Input +/-10V, 0-10V, 0/4-20mA configurable"}
{attribute addProperty Physics "YY"}
{attribute addProperty Id "AI_Standard_Channel_1AT %I*AI_Standard_Channel_A8DF64E310AI_Standard_Channel_2AT %I*AI_Standard_Channel_A8DF64E310WcStateAT %I*WcState_9091E0EB2InfoDataAT %I*InfoData_32EB74EA10"}
{attribute addProperty CRC "2854279291"}
{attribute addProperty Size "32"}
TYPE EP3162_AA20D87B EXTENDS EtcSlaveBoxBase_77A0E4A7 :
STRUCT
	{attribute addProperty Name "AI_Standard_Channel_1"}
	AI_Standard_Channel_1 : AI_Standard_Channel_A8DF64E3;
	{attribute addProperty Name "AI_Standard_Channel_2"}
	AI_Standard_Channel_2 : AI_Standard_Channel_A8DF64E3;
	{attribute addProperty Name "WcState"}
	WcState : WcState_9091E0EB;
	{attribute addProperty Name "InfoData"}
	InfoData : InfoData_32EB74EA;
END_STRUCT
END_TYPE

// ---- DUTs/IO/Boxes/EP3162_C396CC55.TcDUT
{attribute 'GeneratedUsingTerminal: EP3162-1002-0017'}
{attribute addProperty BoxType "EP3162-1002-0017"}
{attribute addProperty Description "EP3162-1002 2Ch. Ana. Input +/-10V, 0-10V, configurable"}
{attribute addProperty Physics "YY"}
{attribute addProperty Id "AI_Standard_Channel_1AT %I*AI_Standard_Channel_A8DF64E310AI_Standard_Channel_2AT %I*AI_Standard_Channel_A8DF64E310DO_OutputsAT %Q*DO_Outputs_C0F4C3832WcStateAT %I*WcState_9091E0EB2InfoDataAT %I*InfoData_32EB74EA10"}
{attribute addProperty CRC "3281439829"}
{attribute addProperty Size "34"}
TYPE EP3162_C396CC55 EXTENDS EtcSlaveBoxBase_77A0E4A7 :
STRUCT
	{attribute addProperty Name "AI_Standard_Channel_1"}
	AI_Standard_Channel_1 : AI_Standard_Channel_A8DF64E3;
	{attribute addProperty Name "AI_Standard_Channel_2"}
	AI_Standard_Channel_2 : AI_Standard_Channel_A8DF64E3;
	{attribute addProperty Name "DO_Outputs"}
	DO_Outputs : DO_Outputs_C0F4C383;
	{attribute addProperty Name "WcState"}
	WcState : WcState_9091E0EB;
	{attribute addProperty Name "InfoData"}
	InfoData : InfoData_32EB74EA;
END_STRUCT
END_TYPE

// ---- DUTs/IO/Boxes/EP3174_C4269E32.TcDUT
{attribute 'GeneratedUsingTerminal: EP3174-0002-0016'}
{attribute addProperty BoxType "EP3174-0002-0016"}
{attribute addProperty Description "EP3174-0002 4Ch. Ana. Input +/-10V, 0-10V, 0/4-20mA configurable"}
{attribute addProperty Physics "YY"}
{attribute addProperty Id "AI_Standard_Channel_1AT %I*AI_Standard_Channel_4A3944819AI_Standard_Channel_2AT %I*AI_Standard_Channel_4A3944819AI_Standard_Channel_3AT %I*AI_Standard_Channel_4A3944819AI_Standard_Channel_4AT %I*AI_Standard_Channel_4A3944819WcStateAT %I*WcState_9091E0EB2InfoDataAT %I*InfoData_32EB74EA10"}
{attribute addProperty CRC "3290865202"}
{attribute addProperty Size "48"}
TYPE EP3174_C4269E32 EXTENDS EtcSlaveBoxBase_77A0E4A7 :
STRUCT
	{attribute addProperty Name "AI_Standard_Channel_1"}
	AI_Standard_Channel_1 : AI_Standard_Channel_4A394481;
	{attribute addProperty Name "AI_Standard_Channel_2"}
	AI_Standard_Channel_2 : AI_Standard_Channel_4A394481;
	{attribute addProperty Name "AI_Standard_Channel_3"}
	AI_Standard_Channel_3 : AI_Standard_Channel_4A394481;
	{attribute addProperty Name "AI_Standard_Channel_4"}
	AI_Standard_Channel_4 : AI_Standard_Channel_4A394481;
	{attribute addProperty Name "WcState"}
	WcState : WcState_9091E0EB;
	{attribute addProperty Name "InfoData"}
	InfoData : InfoData_32EB74EA;
END_STRUCT
END_TYPE

// ---- DUTs/IO/Boxes/EP3174_DCC78662.TcDUT
{attribute 'GeneratedUsingTerminal: EP3174-0002-0018'}
{attribute addProperty BoxType "EP3174-0002-0018"}
{attribute addProperty Description "EP3174-0002 4Ch. Ana. Input +/-10V, 0-10V, 0/4-20mA configurable"}
{attribute addProperty Physics "YY"}
{attribute addProperty Id "AI_Standard_Channel_1AT %I*AI_Standard_Channel_A8DF64E310AI_Standard_Channel_2AT %I*AI_Standard_Channel_A8DF64E310AI_Standard_Channel_3AT %I*AI_Standard_Channel_A8DF64E310AI_Standard_Channel_4AT %I*AI_Standard_Channel_A8DF64E310WcStateAT %I*WcState_9091E0EB2InfoDataAT %I*InfoData_32EB74EA10"}
{attribute addProperty CRC "3704063586"}
{attribute addProperty Size "52"}
TYPE EP3174_DCC78662 EXTENDS EtcSlaveBoxBase_77A0E4A7 :
STRUCT
	{attribute addProperty Name "AI_Standard_Channel_1"}
	AI_Standard_Channel_1 : AI_Standard_Channel_A8DF64E3;
	{attribute addProperty Name "AI_Standard_Channel_2"}
	AI_Standard_Channel_2 : AI_Standard_Channel_A8DF64E3;
	{attribute addProperty Name "AI_Standard_Channel_3"}
	AI_Standard_Channel_3 : AI_Standard_Channel_A8DF64E3;
	{attribute addProperty Name "AI_Standard_Channel_4"}
	AI_Standard_Channel_4 : AI_Standard_Channel_A8DF64E3;
	{attribute addProperty Name "WcState"}
	WcState : WcState_9091E0EB;
	{attribute addProperty Name "InfoData"}
	InfoData : InfoData_32EB74EA;
END_STRUCT
END_TYPE

// ---- DUTs/IO/Boxes/EP3182_0BD171D7.TcDUT
{attribute 'GeneratedUsingTerminal: EP3182-1002-0017'}
{attribute addProperty BoxType "EP3182-1002-0017"}
{attribute addProperty Description "EP3182-1002 2Ch. Ana. Input +/-10V, 0-10V, 0/4-20mA configurable, single ended, 2Ch digital output"}
{attribute addProperty Physics "YY"}
{attribute addProperty Id "AI_Standard_Channel_1AT %I*AI_Standard_Channel_4A3944819AI_Standard_Channel_2AT %I*AI_Standard_Channel_4A3944819DO_OutputsAT %Q*DO_Outputs_C0F4C3832WcStateAT %I*WcState_9091E0EB2InfoDataAT %I*InfoData_32EB74EA10"}
{attribute addProperty CRC "198275543"}
{attribute addProperty Size "32"}
TYPE EP3182_0BD171D7 EXTENDS EtcSlaveBoxBase_77A0E4A7 :
STRUCT
	{attribute addProperty Name "AI_Standard_Channel_1"}
	AI_Standard_Channel_1 : AI_Standard_Channel_4A394481;
	{attribute addProperty Name "AI_Standard_Channel_2"}
	AI_Standard_Channel_2 : AI_Standard_Channel_4A394481;
	{attribute addProperty Name "DO_Outputs"}
	DO_Outputs : DO_Outputs_C0F4C383;
	{attribute addProperty Name "WcState"}
	WcState : WcState_9091E0EB;
	{attribute addProperty Name "InfoData"}
	InfoData : InfoData_32EB74EA;
END_STRUCT
END_TYPE

// ---- DUTs/IO/Boxes/EP3182_C396CC55.TcDUT
{attribute 'GeneratedUsingTerminal: EP3182-1002-0018'}
{attribute addProperty BoxType "EP3182-1002-0018"}
{attribute addProperty Description "EP3182-1002 2Ch. Ana. Input +/-10V, 0-10V, 0/4-20mA configurable, single ended, 2Ch digital output"}
{attribute addProperty Physics "YY"}
{attribute addProperty Id "AI_Standard_Channel_1AT %I*AI_Standard_Channel_A8DF64E310AI_Standard_Channel_2AT %I*AI_Standard_Channel_A8DF64E310DO_OutputsAT %Q*DO_Outputs_C0F4C3832WcStateAT %I*WcState_9091E0EB2InfoDataAT %I*InfoData_32EB74EA10"}
{attribute addProperty CRC "3281439829"}
{attribute addProperty Size "34"}
TYPE EP3182_C396CC55 EXTENDS EtcSlaveBoxBase_77A0E4A7 :
STRUCT
	{attribute addProperty Name "AI_Standard_Channel_1"}
	AI_Standard_Channel_1 : AI_Standard_Channel_A8DF64E3;
	{attribute addProperty Name "AI_Standard_Channel_2"}
	AI_Standard_Channel_2 : AI_Standard_Channel_A8DF64E3;
	{attribute addProperty Name "DO_Outputs"}
	DO_Outputs : DO_Outputs_C0F4C383;
	{attribute addProperty Name "WcState"}
	WcState : WcState_9091E0EB;
	{attribute addProperty Name "InfoData"}
	InfoData : InfoData_32EB74EA;
END_STRUCT
END_TYPE

// ---- DUTs/IO/Boxes/EP3184_C4269E32.TcDUT
{attribute 'GeneratedUsingTerminal: EP3184-0002-0016'}
{attribute addProperty BoxType "EP3184-0002-0016"}
{attribute addProperty Description "EP3184-0002 4Ch. Ana. Input +/-10V, 0-10V, 0/4-20mA configurable, single ended"}
{attribute addProperty Physics "YY"}
{attribute addProperty Id "AI_Standard_Channel_1AT %I*AI_Standard_Channel_4A3944819AI_Standard_Channel_2AT %I*AI_Standard_Channel_4A3944819AI_Standard_Channel_3AT %I*AI_Standard_Channel_4A3944819AI_Standard_Channel_4AT %I*AI_Standard_Channel_4A3944819WcStateAT %I*WcState_9091E0EB2InfoDataAT %I*InfoData_32EB74EA10"}
{attribute addProperty CRC "3290865202"}
{attribute addProperty Size "48"}
TYPE EP3184_C4269E32 EXTENDS EtcSlaveBoxBase_77A0E4A7 :
STRUCT
	{attribute addProperty Name "AI_Standard_Channel_1"}
	AI_Standard_Channel_1 : AI_Standard_Channel_4A394481;
	{attribute addProperty Name "AI_Standard_Channel_2"}
	AI_Standard_Channel_2 : AI_Standard_Channel_4A394481;
	{attribute addProperty Name "AI_Standard_Channel_3"}
	AI_Standard_Channel_3 : AI_Standard_Channel_4A394481;
	{attribute addProperty Name "AI_Standard_Channel_4"}
	AI_Standard_Channel_4 : AI_Standard_Channel_4A394481;
	{attribute addProperty Name "WcState"}
	WcState : WcState_9091E0EB;
	{attribute addProperty Name "InfoData"}
	InfoData : InfoData_32EB74EA;
END_STRUCT
END_TYPE

// ---- DUTs/IO/Boxes/EP3184_DCC78662.TcDUT
{attribute 'GeneratedUsingTerminal: EP3184-0002-0017'}
{attribute addProperty BoxType "EP3184-0002-0017"}
{attribute addProperty Description "EP3184-0002 4Ch. Ana. Input +/-10V, 0-10V, 0/4-20mA configurable, single ended"}
{attribute addProperty Physics "YY"}
{attribute addProperty Id "AI_Standard_Channel_1AT %I*AI_Standard_Channel_A8DF64E310AI_Standard_Channel_2AT %I*AI_Standard_Channel_A8DF64E310AI_Standard_Channel_3AT %I*AI_Standard_Channel_A8DF64E310AI_Standard_Channel_4AT %I*AI_Standard_Channel_A8DF64E310WcStateAT %I*WcState_9091E0EB2InfoDataAT %I*InfoData_32EB74EA10"}
{attribute addProperty CRC "3704063586"}
{attribute addProperty Size "52"}
TYPE EP3184_DCC78662 EXTENDS EtcSlaveBoxBase_77A0E4A7 :
STRUCT
	{attribute addProperty Name "AI_Standard_Channel_1"}
	AI_Standard_Channel_1 : AI_Standard_Channel_A8DF64E3;
	{attribute addProperty Name "AI_Standard_Channel_2"}
	AI_Standard_Channel_2 : AI_Standard_Channel_A8DF64E3;
	{attribute addProperty Name "AI_Standard_Channel_3"}
	AI_Standard_Channel_3 : AI_Standard_Channel_A8DF64E3;
	{attribute addProperty Name "AI_Standard_Channel_4"}
	AI_Standard_Channel_4 : AI_Standard_Channel_A8DF64E3;
	{attribute addProperty Name "WcState"}
	WcState : WcState_9091E0EB;
	{attribute addProperty Name "InfoData"}
	InfoData : InfoData_32EB74EA;
END_STRUCT
END_TYPE

// ---- DUTs/IO/Boxes/EP3204_6CD7E119.TcDUT
{attribute 'GeneratedUsingTerminal: EP3204-0002-0017'}
{attribute addProperty BoxType "EP3204-0002-0017"}
{attribute addProperty Description "EP3204-0002 4Ch. Ana. Input PT100 (RTD)"}
{attribute addProperty Physics "YY"}
{attribute addProperty Id "RTD_RTDInputs_Channel_1AT %I*RTD_RTDInputs_Channel_A8DF64E310RTD_RTDInputs_Channel_2AT %I*RTD_RTDInputs_Channel_A8DF64E310RTD_RTDInputs_Channel_3AT %I*RTD_RTDInputs_Channel_A8DF64E310RTD_RTDInputs_Channel_4AT %I*RTD_RTDInputs_Channel_A8DF64E310WcStateAT %I*WcState_9091E0EB2InfoDataAT %I*InfoData_32EB74EA10"}
{attribute addProperty CRC "1826087193"}
{attribute addProperty Size "52"}
TYPE EP3204_6CD7E119 EXTENDS EtcSlaveBoxBase_77A0E4A7 :
STRUCT
	{attribute addProperty Name "RTD_RTDInputs_Channel_1"}
	RTD_RTDInputs_Channel_1 : RTD_RTDInputs_Channel_A8DF64E3;
	{attribute addProperty Name "RTD_RTDInputs_Channel_2"}
	RTD_RTDInputs_Channel_2 : RTD_RTDInputs_Channel_A8DF64E3;
	{attribute addProperty Name "RTD_RTDInputs_Channel_3"}
	RTD_RTDInputs_Channel_3 : RTD_RTDInputs_Channel_A8DF64E3;
	{attribute addProperty Name "RTD_RTDInputs_Channel_4"}
	RTD_RTDInputs_Channel_4 : RTD_RTDInputs_Channel_A8DF64E3;
	{attribute addProperty Name "WcState"}
	WcState : WcState_9091E0EB;
	{attribute addProperty Name "InfoData"}
	InfoData : InfoData_32EB74EA;
END_STRUCT
END_TYPE

// ---- DUTs/IO/Boxes/EP3204_AB25C3AC.TcDUT
{attribute 'GeneratedUsingTerminal: EP3204-0002-0021'}
{attribute addProperty BoxType "EP3204-0002-0021"}
{attribute addProperty Description "EP3204-0002 4Ch. Ana. Input PT100 (RTD)"}
{attribute addProperty Physics "YY"}
{attribute addProperty Id "RTD_RTDInputs_Channel_1AT %I*AI_Standard_Channel_4A3944819RTD_RTDInputs_Channel_2AT %I*AI_Standard_Channel_4A3944819RTD_RTDInputs_Channel_3AT %I*AI_Standard_Channel_4A3944819RTD_RTDInputs_Channel_4AT %I*AI_Standard_Channel_4A3944819WcStateAT %I*WcState_9091E0EB2InfoDataAT %I*InfoData_32EB74EA10"}
{attribute addProperty CRC "2871378860"}
{attribute addProperty Size "48"}
TYPE EP3204_AB25C3AC EXTENDS EtcSlaveBoxBase_77A0E4A7 :
STRUCT
	{attribute addProperty Name "RTD_RTDInputs_Channel_1"}
	RTD_RTDInputs_Channel_1 : AI_Standard_Channel_4A394481;
	{attribute addProperty Name "RTD_RTDInputs_Channel_2"}
	RTD_RTDInputs_Channel_2 : AI_Standard_Channel_4A394481;
	{attribute addProperty Name "RTD_RTDInputs_Channel_3"}
	RTD_RTDInputs_Channel_3 : AI_Standard_Channel_4A394481;
	{attribute addProperty Name "RTD_RTDInputs_Channel_4"}
	RTD_RTDInputs_Channel_4 : AI_Standard_Channel_4A394481;
	{attribute addProperty Name "WcState"}
	WcState : WcState_9091E0EB;
	{attribute addProperty Name "InfoData"}
	InfoData : InfoData_32EB74EA;
END_STRUCT
END_TYPE

// ---- DUTs/IO/Boxes/EP3314_1CEB931C.TcDUT
{attribute 'GeneratedUsingTerminal: EP3314-0002-0016'}
{attribute addProperty BoxType "EP3314-0002-0016"}
{attribute addProperty Description "EP3314-0002 4Ch. Ana. Input Thermocouple (TC)"}
{attribute addProperty Physics "YY"}
{attribute addProperty Id "TC_TCInputs_Channel_1AT %I*TC_TCInputs_Channel_A8DF64E310TC_TCInputs_Channel_2AT %I*TC_TCInputs_Channel_A8DF64E310TC_TCInputs_Channel_3AT %I*TC_TCInputs_Channel_A8DF64E310TC_TCInputs_Channel_4AT %I*TC_TCInputs_Channel_A8DF64E310WcStateAT %I*WcState_9091E0EB2InfoDataAT %I*InfoData_32EB74EA10"}
{attribute addProperty CRC "485200668"}
{attribute addProperty Size "52"}
TYPE EP3314_1CEB931C EXTENDS EtcSlaveBoxBase_77A0E4A7 :
STRUCT
	{attribute addProperty Name "TC_TCInputs_Channel_1"}
	TC_TCInputs_Channel_1 : TC_TCInputs_Channel_A8DF64E3;
	{attribute addProperty Name "TC_TCInputs_Channel_2"}
	TC_TCInputs_Channel_2 : TC_TCInputs_Channel_A8DF64E3;
	{attribute addProperty Name "TC_TCInputs_Channel_3"}
	TC_TCInputs_Channel_3 : TC_TCInputs_Channel_A8DF64E3;
	{attribute addProperty Name "TC_TCInputs_Channel_4"}
	TC_TCInputs_Channel_4 : TC_TCInputs_Channel_A8DF64E3;
	{attribute addProperty Name "WcState"}
	WcState : WcState_9091E0EB;
	{attribute addProperty Name "InfoData"}
	InfoData : InfoData_32EB74EA;
END_STRUCT
END_TYPE

// ---- DUTs/IO/Boxes/EP3314_E65CDB1C.TcDUT
{attribute 'GeneratedUsingTerminal: EP3314-0002-0019'}
{attribute addProperty BoxType "EP3314-0002-0019"}
{attribute addProperty Description "EP3314-0002 4Ch. Ana. Input Thermocouple (TC)"}
{attribute addProperty Physics "YY"}
{attribute addProperty Id "TC_Inputs_Channel_1AT %I*AI_Standard_Channel_4A3944819TC_Inputs_Channel_2AT %I*AI_Standard_Channel_4A3944819TC_Inputs_Channel_3AT %I*AI_Standard_Channel_4A3944819TC_Inputs_Channel_4AT %I*AI_Standard_Channel_4A3944819WcStateAT %I*WcState_9091E0EB2InfoDataAT %I*InfoData_32EB74EA10"}
{attribute addProperty CRC "3864845084"}
{attribute addProperty Size "48"}
TYPE EP3314_E65CDB1C EXTENDS EtcSlaveBoxBase_77A0E4A7 :
STRUCT
	{attribute addProperty Name "TC_Inputs_Channel_1"}
	TC_Inputs_Channel_1 : AI_Standard_Channel_4A394481;
	{attribute addProperty Name "TC_Inputs_Channel_2"}
	TC_Inputs_Channel_2 : AI_Standard_Channel_4A394481;
	{attribute addProperty Name "TC_Inputs_Channel_3"}
	TC_Inputs_Channel_3 : AI_Standard_Channel_4A394481;
	{attribute addProperty Name "TC_Inputs_Channel_4"}
	TC_Inputs_Channel_4 : AI_Standard_Channel_4A394481;
	{attribute addProperty Name "WcState"}
	WcState : WcState_9091E0EB;
	{attribute addProperty Name "InfoData"}
	InfoData : InfoData_32EB74EA;
END_STRUCT
END_TYPE

// ---- DUTs/IO/Boxes/EP3351_6847F283.TcDUT
{attribute 'GeneratedUsingTerminal: EP3351-2022-0016'}
{attribute addProperty BoxType "EP3351-2022-0016"}
{attribute addProperty Description "EP3351-2022 1Ch. Ana Input Resistor Bridge, Diff. 16bit "}
{attribute addProperty Physics "YY"}
{attribute addProperty Id "AIBridge_InputsAT %I*AIBridge_Inputs_555AA1E89AISupply_InputsAT %I*AISupply_Inputs_555AA1E89WcStateAT %I*WcState_9091E0EB2InfoDataAT %I*InfoData_32EB74EA10"}
{attribute addProperty CRC "1749545603"}
{attribute addProperty Size "30"}
TYPE EP3351_6847F283 EXTENDS EtcSlaveBoxBase_77A0E4A7 :
STRUCT
	{attribute addProperty Name "AIBridge_Inputs"}
	AIBridge_Inputs : AIBridge_Inputs_555AA1E8;
	{attribute addProperty Name "AISupply_Inputs"}
	AISupply_Inputs : AISupply_Inputs_555AA1E8;
	{attribute addProperty Name "WcState"}
	WcState : WcState_9091E0EB;
	{attribute addProperty Name "InfoData"}
	InfoData : InfoData_32EB74EA;
END_STRUCT
END_TYPE

// ---- DUTs/IO/Boxes/EP3356_1EAAA6FF.TcDUT
{attribute 'GeneratedUsingTerminal: EP3356-0022-0016'}
{attribute addProperty BoxType "EP3356-0022-0016"}
{attribute addProperty Description "EP3356-0022 1Ch. Ana. Input Resistor Bridge Terminal, 24bit, High Precision"}
{attribute addProperty Physics "YY"}
{attribute addProperty Id "RMB_StatusAT %I*RMB_Status_C0E100AA7RMB_Value_INT32AT %I*RMB_Value_INT_E9189C4B4RMB_ControlAT %Q*RMB_Control_CC49845C5WcStateAT %I*WcState_9091E0EB2InfoDataAT %I*InfoData_32EB74EA10"}
{attribute addProperty CRC "514500351"}
{attribute addProperty Size "28"}
TYPE EP3356_1EAAA6FF EXTENDS EtcSlaveBoxBase_77A0E4A7 :
STRUCT
	{attribute addProperty Name "RMB_Status"}
	RMB_Status : RMB_Status_C0E100AA;
	{attribute addProperty Name "RMB_Value_INT32"}
	RMB_Value_INT32 : RMB_Value_INT_E9189C4B;
	{attribute addProperty Name "RMB_Control"}
	RMB_Control : RMB_Control_CC49845C;
	{attribute addProperty Name "WcState"}
	WcState : WcState_9091E0EB;
	{attribute addProperty Name "InfoData"}
	InfoData : InfoData_32EB74EA;
END_STRUCT
END_TYPE

// ---- DUTs/IO/Boxes/EP3632_E2B98A5C.TcDUT
{attribute 'GeneratedUsingTerminal: EP3632-0001-0016'}
{attribute addProperty BoxType "EP3632-0001-0016"}
{attribute addProperty Description "EP3632-0001 2Ch. IEPE Sensor"}
{attribute addProperty Physics "YY"}
{attribute addProperty Id "Ch1_StatusAT %I*Ch1_Status_758244858Ch1_Sample_0AT %I*Ch1_Sample_A71DD5012Ch1_Sample_1AT %I*Ch1_Sample_A71DD5012Ch1_Sample_2AT %I*Ch1_Sample_A71DD5012Ch1_Sample_3AT %I*Ch1_Sample_A71DD5012Ch1_Sample_4AT %I*Ch1_Sample_A71DD5012Ch1_Sample_5AT %I*Ch1_Sample_A71DD5012Ch1_Sample_6AT %I*Ch1_Sample_A71DD5012Ch1_Sample_7AT %I*Ch1_Sample_A71DD5012Ch1_Sample_8AT %I*Ch1_Sample_A71DD5012Ch1_Sample_9AT %I*Ch1_Sample_A71DD5012Ch2_StatusAT %I*Ch2_Status_758244858Ch2_Sample_0AT %I*Ch2_Sample_9F6886E62Ch2_Sample_1AT %I*Ch2_Sample_9F6886E62Ch2_Sample_2AT %I*Ch2_Sample_9F6886E62Ch2_Sample_3AT %I*Ch2_Sample_9F6886E62Ch2_Sample_4AT %I*Ch2_Sample_9F6886E62Ch2_Sample_5AT %I*Ch2_Sample_9F6886E62Ch2_Sample_6AT %I*Ch2_Sample_9F6886E62Ch2_Sample_7AT %I*Ch2_Sample_9F6886E62Ch2_Sample_8AT %I*Ch2_Sample_9F6886E62Ch2_Sample_9AT %I*Ch2_Sample_9F6886E62NextSync1TimeAT %I*NextSync1Time_9AFDC2758Sample_CountAT %I*Sample_Count_EA88CAD92WcStateAT %I*WcState_9091E0EB2InfoDataAT %I*InfoData_BEF6B88E18"}
{attribute addProperty CRC "3803810396"}
{attribute addProperty Size "86"}
TYPE EP3632_E2B98A5C EXTENDS EtcSlaveBoxBase_77A0E4A7 :
STRUCT
	{attribute addProperty Name "Ch1_Status"}
	Ch1_Status : Ch1_Status_75824485;
	{attribute addProperty Name "Ch1_Sample_0"}
	Ch1_Sample_0 : Ch1_Sample_A71DD501;
	{attribute addProperty Name "Ch1_Sample_1"}
	Ch1_Sample_1 : Ch1_Sample_A71DD501;
	{attribute addProperty Name "Ch1_Sample_2"}
	Ch1_Sample_2 : Ch1_Sample_A71DD501;
	{attribute addProperty Name "Ch1_Sample_3"}
	Ch1_Sample_3 : Ch1_Sample_A71DD501;
	{attribute addProperty Name "Ch1_Sample_4"}
	Ch1_Sample_4 : Ch1_Sample_A71DD501;
	{attribute addProperty Name "Ch1_Sample_5"}
	Ch1_Sample_5 : Ch1_Sample_A71DD501;
	{attribute addProperty Name "Ch1_Sample_6"}
	Ch1_Sample_6 : Ch1_Sample_A71DD501;
	{attribute addProperty Name "Ch1_Sample_7"}
	Ch1_Sample_7 : Ch1_Sample_A71DD501;
	{attribute addProperty Name "Ch1_Sample_8"}
	Ch1_Sample_8 : Ch1_Sample_A71DD501;
	{attribute addProperty Name "Ch1_Sample_9"}
	Ch1_Sample_9 : Ch1_Sample_A71DD501;
	{attribute addProperty Name "Ch2_Status"}
	Ch2_Status : Ch2_Status_75824485;
	{attribute addProperty Name "Ch2_Sample_0"}
	Ch2_Sample_0 : Ch2_Sample_9F6886E6;
	{attribute addProperty Name "Ch2_Sample_1"}
	Ch2_Sample_1 : Ch2_Sample_9F6886E6;
	{attribute addProperty Name "Ch2_Sample_2"}
	Ch2_Sample_2 : Ch2_Sample_9F6886E6;
	{attribute addProperty Name "Ch2_Sample_3"}
	Ch2_Sample_3 : Ch2_Sample_9F6886E6;
	{attribute addProperty Name "Ch2_Sample_4"}
	Ch2_Sample_4 : Ch2_Sample_9F6886E6;
	{attribute addProperty Name "Ch2_Sample_5"}
	Ch2_Sample_5 : Ch2_Sample_9F6886E6;
	{attribute addProperty Name "Ch2_Sample_6"}
	Ch2_Sample_6 : Ch2_Sample_9F6886E6;
	{attribute addProperty Name "Ch2_Sample_7"}
	Ch2_Sample_7 : Ch2_Sample_9F6886E6;
	{attribute addProperty Name "Ch2_Sample_8"}
	Ch2_Sample_8 : Ch2_Sample_9F6886E6;
	{attribute addProperty Name "Ch2_Sample_9"}
	Ch2_Sample_9 : Ch2_Sample_9F6886E6;
	{attribute addProperty Name "NextSync1Time"}
	NextSync1Time : NextSync1Time_9AFDC275;
	{attribute addProperty Name "Sample_Count"}
	Sample_Count : Sample_Count_EA88CAD9;
	{attribute addProperty Name "WcState"}
	WcState : WcState_9091E0EB;
	{attribute addProperty Name "InfoData"}
	InfoData : InfoData_BEF6B88E;
END_STRUCT
END_TYPE

// ---- DUTs/IO/Boxes/EP3744_315C92D4.TcDUT
{attribute 'GeneratedUsingTerminal: EP3744-0041-0016'}
{attribute addProperty BoxType "EP3744-0041-0016"}
{attribute addProperty Description "EP3744-0041 5Ch. Absolute Pressure 6Ch. Dig. Input 10us 2Ch. Dig. Output 24V 0,5A M8"}
{attribute addProperty Physics "YY"}
{attribute addProperty Id "DIG_InputsAT %I*DIG_Inputs_697E0EF26AI_Inputs_Channel_1AT %I*AI_Inputs_Channel_4521310411AI_Inputs_Channel_2AT %I*AI_Inputs_Channel_4521310411AI_Inputs_Channel_3AT %I*AI_Inputs_Channel_4521310411AI_Inputs_Channel_4AT %I*AI_Inputs_Channel_4521310411DEV_Inputs_DeviceAT %I*DEV_Inputs_Device_5F4E175E5DIG_OutputsAT %Q*DIG_Outputs_DE230DD52DEV_Outputs_DeviceAT %Q*DEV_Outputs_Device_59FFD2471WcStateAT %I*WcState_9091E0EB2InfoDataAT %I*InfoData_32EB74EA10"}
{attribute addProperty CRC "828150484"}
{attribute addProperty Size "70"}
TYPE EP3744_315C92D4 EXTENDS EtcSlaveBoxBase_77A0E4A7 :
STRUCT
	{attribute addProperty Name "DIG_Inputs"}
	DIG_Inputs : DIG_Inputs_697E0EF2;
	{attribute addProperty Name "AI_Inputs_Channel_1"}
	AI_Inputs_Channel_1 : AI_Inputs_Channel_45213104;
	{attribute addProperty Name "AI_Inputs_Channel_2"}
	AI_Inputs_Channel_2 : AI_Inputs_Channel_45213104;
	{attribute addProperty Name "AI_Inputs_Channel_3"}
	AI_Inputs_Channel_3 : AI_Inputs_Channel_45213104;
	{attribute addProperty Name "AI_Inputs_Channel_4"}
	AI_Inputs_Channel_4 : AI_Inputs_Channel_45213104;
	{attribute addProperty Name "DEV_Inputs_Device"}
	DEV_Inputs_Device : DEV_Inputs_Device_5F4E175E;
	{attribute addProperty Name "DIG_Outputs"}
	DIG_Outputs : DIG_Outputs_DE230DD5;
	{attribute addProperty Name "DEV_Outputs_Device"}
	DEV_Outputs_Device : DEV_Outputs_Device_59FFD247;
	{attribute addProperty Name "WcState"}
	WcState : WcState_9091E0EB;
	{attribute addProperty Name "InfoData"}
	InfoData : InfoData_32EB74EA;
END_STRUCT
END_TYPE

// ---- DUTs/IO/Boxes/EP3752_C992DA1B.TcDUT
{attribute 'GeneratedUsingTerminal: EP3752-0000-0017'}
{attribute addProperty BoxType "EP3752-0000-0017"}
{attribute addProperty Description "EP3752-0000 Acceleration Sensor"}
{attribute addProperty Physics "YY"}
{attribute addProperty Id "AI_Inputs_Channel_1AT %I*AI_Inputs_Channel_5A86716D5AI_Inputs_Channel_2AT %I*AI_Inputs_Channel_5A86716D5AI_Inputs_Channel_3AT %I*AI_Inputs_Channel_5A86716D5AI_Inputs_Channel_4AT %I*AI_Inputs_Channel_5A86716D5AI_Inputs_Channel_5AT %I*AI_Inputs_Channel_5A86716D5AI_Inputs_Channel_6AT %I*AI_Inputs_Channel_5A86716D5WcStateAT %I*WcState_9091E0EB2InfoDataAT %I*InfoData_32EB74EA10"}
{attribute addProperty CRC "3381844507"}
{attribute addProperty Size "42"}
TYPE EP3752_C992DA1B EXTENDS EtcSlaveBoxBase_77A0E4A7 :
STRUCT
	{attribute addProperty Name "AI_Inputs_Channel_1"}
	AI_Inputs_Channel_1 : AI_Inputs_Channel_5A86716D;
	{attribute addProperty Name "AI_Inputs_Channel_2"}
	AI_Inputs_Channel_2 : AI_Inputs_Channel_5A86716D;
	{attribute addProperty Name "AI_Inputs_Channel_3"}
	AI_Inputs_Channel_3 : AI_Inputs_Channel_5A86716D;
	{attribute addProperty Name "AI_Inputs_Channel_4"}
	AI_Inputs_Channel_4 : AI_Inputs_Channel_5A86716D;
	{attribute addProperty Name "AI_Inputs_Channel_5"}
	AI_Inputs_Channel_5 : AI_Inputs_Channel_5A86716D;
	{attribute addProperty Name "AI_Inputs_Channel_6"}
	AI_Inputs_Channel_6 : AI_Inputs_Channel_5A86716D;
	{attribute addProperty Name "WcState"}
	WcState : WcState_9091E0EB;
	{attribute addProperty Name "InfoData"}
	InfoData : InfoData_32EB74EA;
END_STRUCT
END_TYPE

// ---- DUTs/IO/Boxes/EP4174_AB92710E.TcDUT
{attribute 'GeneratedUsingTerminal: EP4174-0002-0016'}
{attribute addProperty BoxType "EP4174-0002-0016"}
{attribute addProperty Description "EP4174-0002 4Ch. Ana. Output +/-10V, 0-10V, 0/4-20mA configurable"}
{attribute addProperty Physics "YY"}
{attribute addProperty Id "AO_Outputs_Channel_1AT %Q*AO_Output_Channel_BA7EBB7C2AO_Outputs_Channel_2AT %Q*AO_Output_Channel_BA7EBB7C2AO_Outputs_Channel_3AT %Q*AO_Output_Channel_BA7EBB7C2AO_Outputs_Channel_4AT %Q*AO_Output_Channel_BA7EBB7C2WcStateAT %I*WcState_0B2B16F91InfoDataAT %I*InfoData_32EB74EA10"}
{attribute addProperty CRC "2878501134"}
{attribute addProperty Size "19"}
TYPE EP4174_AB92710E EXTENDS EtcSlaveBoxBase_77A0E4A7 :
STRUCT
	{attribute addProperty Name "AO_Outputs_Channel_1"}
	AO_Outputs_Channel_1 : AO_Output_Channel_BA7EBB7C;
	{attribute addProperty Name "AO_Outputs_Channel_2"}
	AO_Outputs_Channel_2 : AO_Output_Channel_BA7EBB7C;
	{attribute addProperty Name "AO_Outputs_Channel_3"}
	AO_Outputs_Channel_3 : AO_Output_Channel_BA7EBB7C;
	{attribute addProperty Name "AO_Outputs_Channel_4"}
	AO_Outputs_Channel_4 : AO_Output_Channel_BA7EBB7C;
	{attribute addProperty Name "WcState"}
	WcState : WcState_0B2B16F9;
	{attribute addProperty Name "InfoData"}
	InfoData : InfoData_32EB74EA;
END_STRUCT
END_TYPE

// ---- DUTs/IO/Boxes/EP4314_454AD8BA.TcDUT
{attribute 'GeneratedUsingTerminal: EP4314-1002-0016'}
{attribute addProperty BoxType "EP4314-1002-0016"}
{attribute addProperty Description "EP4314-1002 2Ch. Ana. Input -20/0/4-20mA; 2Ch. Ana. Output -20/0/4-20mA configurable"}
{attribute addProperty Physics "YY"}
{attribute addProperty Id "DI_InputsAT %I*DI_Inputs_1F3A93254AI_Standard_Channel_1AT %I*AI_Standard_Channel_4A3944819AI_Standard_Channel_2AT %I*AI_Standard_Channel_4A3944819AO_Standard_Channel_1AT %Q*AO_Output_Channel_BA7EBB7C2AO_Standard_Channel_2AT %Q*AO_Output_Channel_BA7EBB7C2WcStateAT %I*WcState_9091E0EB2InfoDataAT %I*InfoData_32EB74EA10"}
{attribute addProperty CRC "1162533050"}
{attribute addProperty Size "38"}
TYPE EP4314_454AD8BA EXTENDS EtcSlaveBoxBase_77A0E4A7 :
STRUCT
	{attribute addProperty Name "DI_Inputs"}
	DI_Inputs : DI_Inputs_1F3A9325;
	{attribute addProperty Name "AI_Standard_Channel_1"}
	AI_Standard_Channel_1 : AI_Standard_Channel_4A394481;
	{attribute addProperty Name "AI_Standard_Channel_2"}
	AI_Standard_Channel_2 : AI_Standard_Channel_4A394481;
	{attribute addProperty Name "AO_Standard_Channel_1"}
	AO_Standard_Channel_1 : AO_Output_Channel_BA7EBB7C;
	{attribute addProperty Name "AO_Standard_Channel_2"}
	AO_Standard_Channel_2 : AO_Output_Channel_BA7EBB7C;
	{attribute addProperty Name "WcState"}
	WcState : WcState_9091E0EB;
	{attribute addProperty Name "InfoData"}
	InfoData : InfoData_32EB74EA;
END_STRUCT
END_TYPE

// ---- DUTs/IO/Boxes/EP4374_D4EA2234.TcDUT
{attribute 'GeneratedUsingTerminal: EP4374-0002-0016'}
{attribute addProperty BoxType "EP4374-0002-0016"}
{attribute addProperty Description "EP4374-0002 2Ch. Ana. Input +/-10V, 0-10V, 0/4-20mA configurable; 2Ch. Ana. Output +/-10V, 0-10V, 0/4-20mA configurable"}
{attribute addProperty Physics "YY"}
{attribute addProperty Id "AI_TxPDO_Map_Standard_Channel_1AT %I*AI_TxPDO_Map_Standard_Channel_A8DF64E310AI_TxPDO_Map_Standard_Channel_2AT %I*AI_TxPDO_Map_Standard_Channel_A8DF64E310AO_RxPDO_Map_Channel_3AT %Q*AO_Output_Channel_BA7EBB7C2AO_RxPDO_Map_Channel_4AT %Q*AO_Output_Channel_BA7EBB7C2WcStateAT %I*WcState_9091E0EB2InfoDataAT %I*InfoData_32EB74EA10"}
{attribute addProperty CRC "3572113972"}
{attribute addProperty Size "36"}
TYPE EP4374_D4EA2234 EXTENDS EtcSlaveBoxBase_77A0E4A7 :
STRUCT
	{attribute addProperty Name "AI_TxPDO_Map_Standard_Channel_1"}
	AI_TxPDO_Map_Standard_Channel_1 : AI_TxPDO_Map_Standard_Channel_A8DF64E3;
	{attribute addProperty Name "AI_TxPDO_Map_Standard_Channel_2"}
	AI_TxPDO_Map_Standard_Channel_2 : AI_TxPDO_Map_Standard_Channel_A8DF64E3;
	{attribute addProperty Name "AO_RxPDO_Map_Channel_3"}
	AO_RxPDO_Map_Channel_3 : AO_Output_Channel_BA7EBB7C;
	{attribute addProperty Name "AO_RxPDO_Map_Channel_4"}
	AO_RxPDO_Map_Channel_4 : AO_Output_Channel_BA7EBB7C;
	{attribute addProperty Name "WcState"}
	WcState : WcState_9091E0EB;
	{attribute addProperty Name "InfoData"}
	InfoData : InfoData_32EB74EA;
END_STRUCT
END_TYPE

